LIN {X 0,Y 398.84,Z 465.372,A -85,B 0,C 180,E1 -19980.431,E2 -19980.431} C_VEL
LIN {X 0,Y 402.252,Z 471.24,A -85,B 0,C 180,E1 -19988.433,E2 -19988.433} C_VEL
LIN {X 0,Y 405.408,Z 476.012,A -85,B 0,C 180,E1 -19991.524,E2 -19991.524} C_VEL
LIN {X 0,Y 406.667,Z 477.45,A -85,B 0,C 180,E1 -19992.496,E2 -19992.496} C_VEL
LIN {X 0,Y 410.077,Z 482.026,A -85,B 0,C 180,E1 -19994.834,E2 -19994.834} C_VEL
LIN {X 0,Y 414.526,Z 488.461,A -85,B 0,C 180,E1 -19997.404,E2 -19997.404} C_VEL
LIN {X 0,Y 418.678,Z 494.427,A -85,B 0,C 180,E1 -19999.461,E2 -19999.461} C_VEL
LIN {X 0,Y 424.057,Z 502.276,A -85,B 0,C 180,E1 -20001.8,E2 -20001.8} C_VEL
LIN {X 0,Y 431.293,Z 513.364,A -85,B 0,C 180,E1 -20004.555,E2 -20004.555} C_VEL
LIN {X 0,Y 439.263,Z 526.549,A -85,B 0,C 180,E1 -20007.228,E2 -20007.228} C_VEL
LIN {X 0,Y 440.254,Z 528.583,A -85,B 0,C 180,E1 -20007.551,E2 -20007.551} C_VEL
LIN {X 0,Y 424.232,Z 746.146,A -85,B 0,C 180,E1 -20011.089,E2 -20011.089} C_VEL
LIN {X 0,Y 420.857,Z 772.773,A -85,B 0,C 180,E1 -20011.685,E2 -20011.685} C_VEL
LIN {X 0,Y 417.276,Z 793.387,A -85,B 0,C 180,E1 -20012.304,E2 -20012.304} C_VEL
LIN {X 0,Y 412.24,Z 816.827,A -85,B 0,C 180,E1 -20013.197,E2 -20013.197} C_VEL
LIN {X 0,Y 406.718,Z 837.855,A -85,B 0,C 180,E1 -20014.207,E2 -20014.207} C_VEL
LIN {X 0,Y 400.233,Z 859.541,A -85,B 0,C 180,E1 -20015.469,E2 -20015.469} C_VEL
LIN {X 0,Y 392.916,Z 880.551,A -85,B 0,C 180,E1 -20016.959,E2 -20016.959} C_VEL
LIN {X 0,Y 385.902,Z 898.896,A -85,B 0,C 180,E1 -20018.511,E2 -20018.511} C_VEL
LIN {X 0,Y 376.941,Z 920.104,A -85,B 0,C 180,E1 -20020.654,E2 -20020.654} C_VEL
LIN {X 0,Y 369.253,Z 936.853,A -85,B 0,C 180,E1 -20022.677,E2 -20022.677} C_VEL
LIN {X 0,Y 360.106,Z 955.579,A -85,B 0,C 180,E1 -20025.373,E2 -20025.373} C_VEL
LIN {X 0,Y 352.353,Z 970.558,A -85,B 0,C 180,E1 -20027.956,E2 -20027.956} C_VEL
LIN {X 0,Y 343.98,Z 986.277,A -85,B 0,C 180,E1 -20031.172,E2 -20031.172} C_VEL
LIN {X 0,Y 337.136,Z 998.762,A -85,B 0,C 180,E1 -20034.249,E2 -20034.249} C_VEL
LIN {X 0,Y 330.325,Z 1011.44,A -85,B 0,C 180,E1 -20037.948,E2 -20037.948} C_VEL
LIN {X 0,Y 324.506,Z 1022.333,A -85,B 0,C 180,E1 -20041.873,E2 -20041.873} C_VEL
LIN {X 0,Y 319.832,Z 1031.874,A -85,B 0,C 180,E1 -20046.02,E2 -20046.02} C_VEL
LIN {X 0,Y 316.404,Z 1039.482,A -85,B 0,C 180,E1 -20050.237,E2 -20050.237} C_VEL
LIN {X 0,Y 314.202,Z 1045.368,A -85,B 0,C 180,E1 -20054.306,E2 -20054.306} C_VEL
LIN {X 0,Y 312.792,Z 1050.105,A -85,B 0,C 180,E1 -20058.756,E2 -20058.756} C_VEL
LIN {X 0,Y 312.252,Z 1052.832,A -85,B 0,C 180,E1 -20062.456,E2 -20062.456} C_VEL
LIN {X 0,Y 312.038,Z 1054.512,A -85,B 0,C 180,E1 -20066.142,E2 -20066.142} C_VEL
LIN {X 0,Y 311.99,Z 1055.15,A -85,B 0,C 180,E1 -20070.367,E2 -20070.367} C_VEL
LIN {X 0,Y 312.049,Z 1054.421,A -85,B 0,C 180,E1 -20074.227,E2 -20074.227} C_VEL
LIN {X 0,Y 312.274,Z 1052.681,A -85,B 0,C 180,E1 -20077.914,E2 -20077.914} C_VEL
LIN {X 0,Y 313.002,Z 1049.425,A -85,B 0,C 180,E1 -20082.172,E2 -20082.172} C_VEL
LIN {X 0,Y 314.49,Z 1044.525,A -85,B 0,C 180,E1 -20086.437,E2 -20086.437} C_VEL
LIN {X 0,Y 316.756,Z 1038.711,A -85,B 0,C 180,E1 -20090.359,E2 -20090.359} C_VEL
LIN {X 0,Y 320.659,Z 1030.134,A -85,B 0,C 180,E1 -20094.895,E2 -20094.895} C_VEL
LIN {X 0,Y 324.873,Z 1021.697,A -85,B 0,C 180,E1 -20098.493,E2 -20098.493} C_VEL
LIN {X 0,Y 330.981,Z 1010.268,A -85,B 0,C 180,E1 -20102.53,E2 -20102.53} C_VEL
LIN {X 0,Y 337.538,Z 998.148,A -85,B 0,C 180,E1 -20106.029,E2 -20106.029} C_VEL
LIN {X 0,Y 345.134,Z 984.339,A -85,B 0,C 180,E1 -20109.381,E2 -20109.381} C_VEL
LIN {X 0,Y 353.066,Z 969.367,A -85,B 0,C 180,E1 -20112.378,E2 -20112.378} C_VEL
LIN {X 0,Y 361.534,Z 953.032,A -85,B 0,C 180,E1 -20115.15,E2 -20115.15} C_VEL
LIN {X 0,Y 370.106,Z 935.274,A -85,B 0,C 180,E1 -20117.638,E2 -20117.638} C_VEL
LIN {X 0,Y 378.689,Z 916.559,A -85,B 0,C 180,E1 -20119.853,E2 -20119.853} C_VEL
LIN {X 0,Y 386.864,Z 896.797,A -85,B 0,C 180,E1 -20121.787,E2 -20121.787} C_VEL
LIN {X 0,Y 394.429,Z 876.878,A -85,B 0,C 180,E1 -20123.435,E2 -20123.435} C_VEL
LIN {X 0,Y 401.889,Z 854.633,A -85,B 0,C 180,E1 -20124.94,E2 -20124.94} C_VEL
LIN {X 0,Y 407.945,Z 834.042,A -85,B 0,C 180,E1 -20126.1,E2 -20126.1} C_VEL
LIN {X 0,Y 412.356,Z 817.004,A -85,B 0,C 180,E1 -20126.9,E2 -20126.9} C_VEL
LIN {X 0,Y 413.523,Z 809.94,A -85,B 0,C 180,E1 -20127.317,E2 -20127.317} C_VEL
LIN {X 0,Y 414.052,Z 791.319,A -85,B 0,C 180,E1 -20128.726,E2 -20128.726} C_VEL
LIN {X 0,Y 414.868,Z 785.076,A -85,B 0,C 180,E1 -20129.022,E2 -20129.022} C_VEL
LIN {X 0,Y 418.668,Z 760.478,A -85,B 0,C 180,E1 -20129.662,E2 -20129.662} C_VEL
LIN {X 0,Y 421.165,Z 737.353,A -85,B 0,C 180,E1 -20130.111,E2 -20130.111} C_VEL
LIN {X 0,Y 436.469,Z 532.848,A -85,B 0,C 180,E1 -20133.424,E2 -20133.424} C_VEL
LIN {X 0,Y 428.688,Z 519.811,A -85,B 0,C 180,E1 -20136.129,E2 -20136.129} C_VEL
LIN {X 0,Y 421.455,Z 508.401,A -85,B 0,C 180,E1 -20139.008,E2 -20139.008} C_VEL
LIN {X 0,Y 414.958,Z 498.798,A -85,B 0,C 180,E1 -20142.035,E2 -20142.035} C_VEL
LIN {X 0,Y 411.129,Z 493.354,A -85,B 0,C 180,E1 -20144.121,E2 -20144.121} C_VEL
LIN {X 0,Y 408.284,Z 489.293,A -85,B 0,C 180,E1 -20145.896,E2 -20145.896} C_VEL
LIN {X 0,Y 404.819,Z 484.368,A -85,B 0,C 180,E1 -20148.459,E2 -20148.459} C_VEL
LIN {X 0,Y 401.967,Z 480.55,A -85,B 0,C 180,E1 -20151.128,E2 -20151.128} C_VEL
LIN {X 0,Y 401.27,Z 479.179,A -85,B 0,C 180,E1 -20151.979,E2 -20151.979} C_VEL
LIN {X 0,Y 398.091,Z 474.432,A -85,B 0,C 180,E1 -20159.568,E2 -20159.568} C_VEL
LIN {X 0,Y 398.227,Z 475.335,A -85,B 0,C 180,E1 -20161.871,E2 -20161.871} C_VEL
LIN {X 0,Y 401.485,Z 479.457,A -85,B 0,C 180,E1 -20167.945,E2 -20167.945} C_VEL
LIN {X 0,Y 404.349,Z 483.907,A -85,B 0,C 180,E1 -20170.832,E2 -20170.832} C_VEL
LIN {X 0,Y 405.563,Z 485.403,A -85,B 0,C 180,E1 -20171.808,E2 -20171.808} C_VEL
LIN {X 0,Y 409.4,Z 490.884,A -85,B 0,C 180,E1 -20174.498,E2 -20174.498} C_VEL
LIN {X 0,Y 413.237,Z 496.392,A -85,B 0,C 180,E1 -20176.735,E2 -20176.735} C_VEL
LIN {X 0,Y 417.319,Z 502.3,A -85,B 0,C 180,E1 -20178.8,E2 -20178.8} C_VEL
LIN {X 0,Y 420.643,Z 507.862,A -85,B 0,C 180,E1 -20180.343,E2 -20180.343} C_VEL
LIN {X 0,Y 426.504,Z 518.163,A -85,B 0,C 180,E1 -20182.794,E2 -20182.794} C_VEL
LIN {X 0,Y 434.165,Z 532.67,A -85,B 0,C 180,E1 -20185.62,E2 -20185.62} C_VEL
LIN {X 0,Y 436.3,Z 537.348,A -85,B 0,C 180,E1 -20186.363,E2 -20186.363} C_VEL
LIN {X 0,Y 419.712,Z 757.486,A -85,B 0,C 180,E1 -20189.946,E2 -20189.946} C_VEL
LIN {X 0,Y 416.159,Z 784.326,A -85,B 0,C 180,E1 -20190.522,E2 -20190.522} C_VEL
LIN {X 0,Y 412.096,Z 806.229,A -85,B 0,C 180,E1 -20191.141,E2 -20191.141} C_VEL
LIN {X 0,Y 406.049,Z 832.118,A -85,B 0,C 180,E1 -20192.103,E2 -20192.103} C_VEL
LIN {X 0,Y 400.422,Z 852.323,A -85,B 0,C 180,E1 -20193.057,E2 -20193.057} C_VEL
LIN {X 0,Y 393.151,Z 875.089,A -85,B 0,C 180,E1 -20194.375,E2 -20194.375} C_VEL
LIN {X 0,Y 385.832,Z 895.099,A -85,B 0,C 180,E1 -20195.792,E2 -20195.792} C_VEL
LIN {X 0,Y 377.675,Z 915.487,A -85,B 0,C 180,E1 -20197.512,E2 -20197.512} C_VEL
LIN {X 0,Y 369.176,Z 934.587,A -85,B 0,C 180,E1 -20199.475,E2 -20199.475} C_VEL
LIN {X 0,Y 361.129,Z 951.583,A -85,B 0,C 180,E1 -20201.531,E2 -20201.531} C_VEL
LIN {X 0,Y 351.696,Z 970.23,A -85,B 0,C 180,E1 -20204.238,E2 -20204.238} C_VEL
LIN {X 0,Y 344.137,Z 984.536,A -85,B 0,C 180,E1 -20206.709,E2 -20206.709} C_VEL
LIN {X 0,Y 335.419,Z 1000.614,A -85,B 0,C 180,E1 -20210.007,E2 -20210.007} C_VEL
LIN {X 0,Y 328.07,Z 1013.95,A -85,B 0,C 180,E1 -20213.318,E2 -20213.318} C_VEL
LIN {X 0,Y 321.036,Z 1026.979,A -85,B 0,C 180,E1 -20217.184,E2 -20217.184} C_VEL
LIN {X 0,Y 315.543,Z 1037.501,A -85,B 0,C 180,E1 -20220.999,E2 -20220.999} C_VEL
LIN {X 0,Y 310.872,Z 1047.346,A -85,B 0,C 180,E1 -20225.283,E2 -20225.283} C_VEL
LIN {X 0,Y 307.547,Z 1055.237,A -85,B 0,C 180,E1 -20229.642,E2 -20229.642} C_VEL
LIN {X 0,Y 305.446,Z 1061.626,A -85,B 0,C 180,E1 -20234.039,E2 -20234.039} C_VEL
LIN {X 0,Y 304.32,Z 1066.475,A -85,B 0,C 180,E1 -20238.63,E2 -20238.63} C_VEL
LIN {X 0,Y 303.998,Z 1069.293,A -85,B 0,C 180,E1 -20242.44,E2 -20242.44} C_VEL
LIN {X 0,Y 303.968,Z 1071.08,A -85,B 0,C 180,E1 -20246.417,E2 -20246.417} C_VEL
LIN {X 0,Y 303.99,Z 1071.559,A -85,B 0,C 180,E1 -20250.565,E2 -20250.565} C_VEL
LIN {X 0,Y 303.964,Z 1070.791,A -85,B 0,C 180,E1 -20254.339,E2 -20254.339} C_VEL
LIN {X 0,Y 304.004,Z 1069.044,A -85,B 0,C 180,E1 -20257.94,E2 -20257.94} C_VEL
LIN {X 0,Y 304.413,Z 1065.96,A -85,B 0,C 180,E1 -20261.943,E2 -20261.943} C_VEL
LIN {X 0,Y 305.727,Z 1060.552,A -85,B 0,C 180,E1 -20266.727,E2 -20266.727} C_VEL
LIN {X 0,Y 307.779,Z 1054.575,A -85,B 0,C 180,E1 -20270.739,E2 -20270.739} C_VEL
LIN {X 0,Y 311.571,Z 1045.662,A -85,B 0,C 180,E1 -20275.469,E2 -20275.469} C_VEL
LIN {X 0,Y 316.007,Z 1036.505,A -85,B 0,C 180,E1 -20279.369,E2 -20279.369} C_VEL
LIN {X 0,Y 322.211,Z 1024.682,A -85,B 0,C 180,E1 -20283.53,E2 -20283.53} C_VEL
LIN {X 0,Y 328.76,Z 1012.568,A -85,B 0,C 180,E1 -20287.027,E2 -20287.027} C_VEL
LIN {X 0,Y 336.791,Z 998.007,A -85,B 0,C 180,E1 -20290.555,E2 -20290.555} C_VEL
LIN {X 0,Y 344.827,Z 983.07,A -85,B 0,C 180,E1 -20293.537,E2 -20293.537} C_VEL
LIN {X 0,Y 353.677,Z 966.328,A -85,B 0,C 180,E1 -20296.364,E2 -20296.364} C_VEL
LIN {X 0,Y 362.508,Z 948.447,A -85,B 0,C 180,E1 -20298.851,E2 -20298.851} C_VEL
LIN {X 0,Y 370.86,Z 930.689,A -85,B 0,C 180,E1 -20300.94,E2 -20300.94} C_VEL
LIN {X 0,Y 379.657,Z 910.216,A -85,B 0,C 180,E1 -20302.939,E2 -20302.939} C_VEL
LIN {X 0,Y 387.057,Z 891.531,A -85,B 0,C 180,E1 -20304.463,E2 -20304.463} C_VEL
LIN {X 0,Y 395.358,Z 867.969,A -85,B 0,C 180,E1 -20306.051,E2 -20306.051} C_VEL
LIN {X 0,Y 401.304,Z 848.81,A -85,B 0,C 180,E1 -20307.105,E2 -20307.105} C_VEL
LIN {X 0,Y 407.415,Z 826.398,A -85,B 0,C 180,E1 -20308.121,E2 -20308.121} C_VEL
LIN {X 0,Y 412.484,Z 803.511,A -85,B 0,C 180,E1 -20308.927,E2 -20308.927} C_VEL
LIN {X 0,Y 416.737,Z 779.965,A -85,B 0,C 180,E1 -20309.572,E2 -20309.572} C_VEL
LIN {X 0,Y 419.765,Z 755.051,A -85,B 0,C 180,E1 -20310.084,E2 -20310.084} C_VEL
LIN {X 0,Y 436.13,Z 536.856,A -85,B 0,C 180,E1 -20313.637,E2 -20313.637} C_VEL
LIN {X 0,Y 429.621,Z 524.181,A -85,B 0,C 180,E1 -20315.929,E2 -20315.929} C_VEL
LIN {X 0,Y 423.372,Z 512.779,A -85,B 0,C 180,E1 -20318.381,E2 -20318.381} C_VEL
LIN {X 0,Y 417.521,Z 502.692,A -85,B 0,C 180,E1 -20320.992,E2 -20320.992} C_VEL
LIN {X 0,Y 413.631,Z 497.107,A -85,B 0,C 180,E1 -20322.92,E2 -20322.92} C_VEL
LIN {X 0,Y 411.069,Z 493.426,A -85,B 0,C 180,E1 -20324.336,E2 -20324.336} C_VEL
LIN {X 0,Y 407.99,Z 489,A -85,B 0,C 180,E1 -20326.248,E2 -20326.248} C_VEL
LIN {X 0,Y 404.781,Z 484.386,A -85,B 0,C 180,E1 -20328.602,E2 -20328.602} C_VEL
LIN {X 0,Y 401.616,Z 480.005,A -85,B 0,C 180,E1 -20331.553,E2 -20331.553} C_VEL
LIN {X 0,Y 401.014,Z 479.013,A -85,B 0,C 180,E1 -20332.262,E2 -20332.262} C_VEL
LIN {X 0,Y 397.873,Z 474.137,A -85,B 0,C 180,E1 -20338.848,E2 -20338.848} C_VEL
LIN {X 0,Y 397.864,Z 473.319,A -85,B 0,C 180,E1 -20340.432,E2 -20340.432} C_VEL
LIN {X 0,Y 401.152,Z 479.129,A -85,B 0,C 180,E1 -20348.312,E2 -20348.312} C_VEL
LIN {X 0,Y 404.264,Z 483.898,A -85,B 0,C 180,E1 -20351.412,E2 -20351.412} C_VEL
LIN {X 0,Y 405.406,Z 485.321,A -85,B 0,C 180,E1 -20352.318,E2 -20352.318} C_VEL
LIN {X 0,Y 409.399,Z 490.954,A -85,B 0,C 180,E1 -20355.077,E2 -20355.077} C_VEL
LIN {X 0,Y 413.03,Z 496.212,A -85,B 0,C 180,E1 -20357.178,E2 -20357.178} C_VEL
LIN {X 0,Y 418.41,Z 503.941,A -85,B 0,C 180,E1 -20359.837,E2 -20359.837} C_VEL
LIN {X 0,Y 425.452,Z 514.825,A -85,B 0,C 180,E1 -20362.817,E2 -20362.817} C_VEL
LIN {X 0,Y 432.479,Z 526.228,A -85,B 0,C 180,E1 -20365.396,E2 -20365.396} C_VEL
LIN {X 0,Y 436.287,Z 533.004,A -85,B 0,C 180,E1 -20366.686,E2 -20366.686} C_VEL
LIN {X 0,Y 420.154,Z 746.396,A -85,B 0,C 180,E1 -20370.155,E2 -20370.155} C_VEL
LIN {X 0,Y 416.708,Z 773.001,A -85,B 0,C 180,E1 -20370.748,E2 -20370.748} C_VEL
LIN {X 0,Y 413.075,Z 793.462,A -85,B 0,C 180,E1 -20371.359,E2 -20371.359} C_VEL
LIN {X 0,Y 407.897,Z 817.05,A -85,B 0,C 180,E1 -20372.252,E2 -20372.252} C_VEL
LIN {X 0,Y 402.161,Z 838.378,A -85,B 0,C 180,E1 -20373.275,E2 -20373.275} C_VEL
LIN {X 0,Y 395.294,Z 860.754,A -85,B 0,C 180,E1 -20374.579,E2 -20374.579} C_VEL
LIN {X 0,Y 387.8,Z 881.579,A -85,B 0,C 180,E1 -20376.068,E2 -20376.068} C_VEL
LIN {X 0,Y 380.029,Z 901.307,A -85,B 0,C 180,E1 -20377.755,E2 -20377.755} C_VEL
LIN {X 0,Y 371.133,Z 921.533,A -85,B 0,C 180,E1 -20379.84,E2 -20379.84} C_VEL
LIN {X 0,Y 362.987,Z 938.726,A -85,B 0,C 180,E1 -20381.949,E2 -20381.949} C_VEL
LIN {X 0,Y 353.841,Z 956.717,A -85,B 0,C 180,E1 -20384.594,E2 -20384.594} C_VEL
LIN {X 0,Y 345.862,Z 971.617,A -85,B 0,C 180,E1 -20387.204,E2 -20387.204} C_VEL
LIN {X 0,Y 336.939,Z 987.672,A -85,B 0,C 180,E1 -20390.576,E2 -20390.576} C_VEL
LIN {X 0,Y 330.145,Z 999.611,A -85,B 0,C 180,E1 -20393.586,E2 -20393.586} C_VEL
LIN {X 0,Y 322.986,Z 1012.335,A -85,B 0,C 180,E1 -20397.407,E2 -20397.407} C_VEL
LIN {X 0,Y 317.275,Z 1022.566,A -85,B 0,C 180,E1 -20401.178,E2 -20401.178} C_VEL
LIN {X 0,Y 312.356,Z 1032.094,A -85,B 0,C 180,E1 -20405.409,E2 -20405.409} C_VEL
LIN {X 0,Y 308.722,Z 1039.702,A -85,B 0,C 180,E1 -20409.724,E2 -20409.724} C_VEL
LIN {X 0,Y 306.374,Z 1045.586,A -85,B 0,C 180,E1 -20413.895,E2 -20413.895} C_VEL
LIN {X 0,Y 304.862,Z 1050.321,A -85,B 0,C 180,E1 -20418.459,E2 -20418.459} C_VEL
LIN {X 0,Y 304.276,Z 1053.047,A -85,B 0,C 180,E1 -20422.257,E2 -20422.257} C_VEL
LIN {X 0,Y 304.045,Z 1054.726,A -85,B 0,C 180,E1 -20426.04,E2 -20426.04} C_VEL
LIN {X 0,Y 303.993,Z 1055.363,A -85,B 0,C 180,E1 -20430.377,E2 -20430.377} C_VEL
LIN {X 0,Y 304.056,Z 1054.634,A -85,B 0,C 180,E1 -20434.338,E2 -20434.338} C_VEL
LIN {X 0,Y 304.281,Z 1053.006,A -85,B 0,C 180,E1 -20437.933,E2 -20437.933} C_VEL
LIN {X 0,Y 304.939,Z 1050.106,A -85,B 0,C 180,E1 -20441.922,E2 -20441.922} C_VEL
LIN {X 0,Y 306.595,Z 1044.99,A -85,B 0,C 180,E1 -20446.678,E2 -20446.678} C_VEL
LIN {X 0,Y 308.934,Z 1039.288,A -85,B 0,C 180,E1 -20450.658,E2 -20450.658} C_VEL
LIN {X 0,Y 312.848,Z 1031.149,A -85,B 0,C 180,E1 -20455.156,E2 -20455.156} C_VEL
LIN {X 0,Y 317.426,Z 1022.367,A -85,B 0,C 180,E1 -20459.019,E2 -20459.019} C_VEL
LIN {X 0,Y 323.471,Z 1011.607,A -85,B 0,C 180,E1 -20462.959,E2 -20462.959} C_VEL
LIN {X 0,Y 330.365,Z 999.344,A -85,B 0,C 180,E1 -20466.602,E2 -20466.602} C_VEL
LIN {X 0,Y 338.009,Z 985.993,A -85,B 0,C 180,E1 -20469.936,E2 -20469.936} C_VEL
LIN {X 0,Y 346.544,Z 970.526,A -85,B 0,C 180,E1 -20473.114,E2 -20473.114} C_VEL
LIN {X 0,Y 354.652,Z 955.4,A -85,B 0,C 180,E1 -20475.735,E2 -20475.735} C_VEL
LIN {X 0,Y 363.863,Z 937.14,A -85,B 0,C 180,E1 -20478.37,E2 -20478.37} C_VEL
LIN {X 0,Y 371.824,Z 920.329,A -85,B 0,C 180,E1 -20480.407,E2 -20480.407} C_VEL
LIN {X 0,Y 381.015,Z 899.199,A -85,B 0,C 180,E1 -20482.546,E2 -20482.546} C_VEL
LIN {X 0,Y 388.224,Z 880.852,A -85,B 0,C 180,E1 -20484.097,E2 -20484.097} C_VEL
LIN {X 0,Y 396.047,Z 858.843,A -85,B 0,C 180,E1 -20485.646,E2 -20485.646} C_VEL
LIN {X 0,Y 402.568,Z 837.511,A -85,B 0,C 180,E1 -20486.877,E2 -20486.877} C_VEL
LIN {X 0,Y 408.593,Z 814.944,A -85,B 0,C 180,E1 -20487.945,E2 -20487.945} C_VEL
LIN {X 0,Y 413.602,Z 791.608,A -85,B 0,C 180,E1 -20488.807,E2 -20488.807} C_VEL
LIN {X 0,Y 414.868,Z 785.076,A -85,B 0,C 180,E1 -20489.022,E2 -20489.022} C_VEL
LIN {X 0,Y 415.678,Z 777.754,A -85,B 0,C 180,E1 -20489.363,E2 -20489.363} C_VEL
LIN {X 0,Y 415.335,Z 759.483,A -85,B 0,C 180,E1 -20490.524,E2 -20490.524} C_VEL
LIN {X 0,Y 415.837,Z 752.018,A -85,B 0,C 180,E1 -20490.803,E2 -20490.803} C_VEL
LIN {X 0,Y 419.407,Z 709.213,A -85,B 0,C 180,E1 -20491.53,E2 -20491.53} C_VEL
LIN {X 0,Y 432.567,Z 537.312,A -85,B 0,C 180,E1 -20494.316,E2 -20494.316} C_VEL
LIN {X 0,Y 425.245,Z 524.937,A -85,B 0,C 180,E1 -20496.989,E2 -20496.989} C_VEL
LIN {X 0,Y 418.952,Z 514.929,A -85,B 0,C 180,E1 -20499.607,E2 -20499.607} C_VEL
LIN {X 0,Y 413.188,Z 506.172,A -85,B 0,C 180,E1 -20502.393,E2 -20502.393} C_VEL
LIN {X 0,Y 409.452,Z 500.747,A -85,B 0,C 180,E1 -20504.49,E2 -20504.49} C_VEL
LIN {X 0,Y 406.785,Z 496.87,A -85,B 0,C 180,E1 -20506.206,E2 -20506.206} C_VEL
LIN {X 0,Y 403.499,Z 492.095,A -85,B 0,C 180,E1 -20508.71,E2 -20508.71} C_VEL
LIN {X 0,Y 400.678,Z 488.111,A -85,B 0,C 180,E1 -20511.461,E2 -20511.461} C_VEL
LIN {X 0,Y 400.05,Z 486.996,A -85,B 0,C 180,E1 -20512.243,E2 -20512.243} C_VEL
LIN {X 0,Y 397.115,Z 482.374,A -85,B 0,C 180,E1 -20519.567,E2 -20519.567} C_VEL
LIN {X 0,Y 397.248,Z 483.314,A -85,B 0,C 180,E1 -20521.875,E2 -20521.875} C_VEL
LIN {X 0,Y 400.377,Z 487.415,A -85,B 0,C 180,E1 -20527.823,E2 -20527.823} C_VEL
LIN {X 0,Y 403.208,Z 491.792,A -85,B 0,C 180,E1 -20530.719,E2 -20530.719} C_VEL
LIN {X 0,Y 404.394,Z 493.408,A -85,B 0,C 180,E1 -20531.698,E2 -20531.698} C_VEL
LIN {X 0,Y 407.876,Z 498.429,A -85,B 0,C 180,E1 -20534.191,E2 -20534.191} C_VEL
LIN {X 0,Y 411.628,Z 503.943,A -85,B 0,C 180,E1 -20536.439,E2 -20536.439} C_VEL
LIN {X 0,Y 416.255,Z 510.75,A -85,B 0,C 180,E1 -20538.813,E2 -20538.813} C_VEL
LIN {X 0,Y 423.242,Z 523.257,A -85,B 0,C 180,E1 -20541.954,E2 -20541.954} C_VEL
LIN {X 0,Y 430.627,Z 537.509,A -85,B 0,C 180,E1 -20544.815,E2 -20544.815} C_VEL
LIN {X 0,Y 432.442,Z 541.575,A -85,B 0,C 180,E1 -20545.48,E2 -20545.48} C_VEL
LIN {X 0,Y 415.752,Z 757.4,A -85,B 0,C 180,E1 -20548.989,E2 -20548.989} C_VEL
LIN {X 0,Y 412.138,Z 784.124,A -85,B 0,C 180,E1 -20549.56,E2 -20549.56} C_VEL
LIN {X 0,Y 408.019,Z 805.916,A -85,B 0,C 180,E1 -20550.171,E2 -20550.171} C_VEL
LIN {X 0,Y 402.07,Z 831.01,A -85,B 0,C 180,E1 -20551.091,E2 -20551.091} C_VEL
LIN {X 0,Y 396.315,Z 851.299,A -85,B 0,C 180,E1 -20552.035,E2 -20552.035} C_VEL
LIN {X 0,Y 389.275,Z 873.111,A -85,B 0,C 180,E1 -20553.271,E2 -20553.271} C_VEL
LIN {X 0,Y 381.448,Z 894.071,A -85,B 0,C 180,E1 -20554.737,E2 -20554.737} C_VEL
LIN {X 0,Y 373.304,Z 913.943,A -85,B 0,C 180,E1 -20556.395,E2 -20556.395} C_VEL
LIN {X 0,Y 364.31,Z 933.759,A -85,B 0,C 180,E1 -20558.41,E2 -20558.41} C_VEL
LIN {X 0,Y 356.074,Z 950.663,A -85,B 0,C 180,E1 -20560.448,E2 -20560.448} C_VEL
LIN {X 0,Y 345.996,Z 970.013,A -85,B 0,C 180,E1 -20563.26,E2 -20563.26} C_VEL
LIN {X 0,Y 338.169,Z 984.318,A -85,B 0,C 180,E1 -20565.749,E2 -20565.749} C_VEL
LIN {X 0,Y 329.286,Z 1000.107,A -85,B 0,C 180,E1 -20569.012,E2 -20569.012} C_VEL
LIN {X 0,Y 321.818,Z 1013.087,A -85,B 0,C 180,E1 -20572.26,E2 -20572.26} C_VEL
LIN {X 0,Y 314.654,Z 1025.812,A -85,B 0,C 180,E1 -20576.037,E2 -20576.037} C_VEL
LIN {X 0,Y 308.562,Z 1036.815,A -85,B 0,C 180,E1 -20580.064,E2 -20580.064} C_VEL
LIN {X 0,Y 303.745,Z 1046.326,A -85,B 0,C 180,E1 -20584.245,E2 -20584.245} C_VEL
LIN {X 0,Y 300.09,Z 1054.399,A -85,B 0,C 180,E1 -20588.704,E2 -20588.704} C_VEL
LIN {X 0,Y 297.89,Z 1060.368,A -85,B 0,C 180,E1 -20592.82,E2 -20592.82} C_VEL
LIN {X 0,Y 296.466,Z 1065.765,A -85,B 0,C 180,E1 -20597.732,E2 -20597.732} C_VEL
LIN {X 0,Y 296.016,Z 1068.844,A -85,B 0,C 180,E1 -20601.844,E2 -20601.844} C_VEL
LIN {X 0,Y 295.966,Z 1070.586,A -85,B 0,C 180,E1 -20605.543,E2 -20605.543} C_VEL
LIN {X 0,Y 295.993,Z 1071.349,A -85,B 0,C 180,E1 -20609.419,E2 -20609.419} C_VEL
LIN {X 0,Y 295.969,Z 1070.857,A -85,B 0,C 180,E1 -20613.68,E2 -20613.68} C_VEL
LIN {X 0,Y 295.999,Z 1069.179,A -85,B 0,C 180,E1 -20617.57,E2 -20617.57} C_VEL
LIN {X 0,Y 296.335,Z 1066.401,A -85,B 0,C 180,E1 -20621.483,E2 -20621.483} C_VEL
LIN {X 0,Y 297.444,Z 1061.869,A -85,B 0,C 180,E1 -20626.001,E2 -20626.001} C_VEL
LIN {X 0,Y 299.595,Z 1055.593,A -85,B 0,C 180,E1 -20630.514,E2 -20630.514} C_VEL
LIN {X 0,Y 302.666,Z 1048.514,A -85,B 0,C 180,E1 -20634.598,E2 -20634.598} C_VEL
LIN {X 0,Y 307.826,Z 1038.148,A -85,B 0,C 180,E1 -20639.372,E2 -20639.372} C_VEL
LIN {X 0,Y 313.181,Z 1028.252,A -85,B 0,C 180,E1 -20643.089,E2 -20643.089} C_VEL
LIN {X 0,Y 320.721,Z 1014.918,A -85,B 0,C 180,E1 -20647.216,E2 -20647.216} C_VEL
LIN {X 0,Y 327.616,Z 1002.826,A -85,B 0,C 180,E1 -20650.318,E2 -20650.318} C_VEL
LIN {X 0,Y 336.296,Z 987.588,A -85,B 0,C 180,E1 -20653.613,E2 -20653.613} C_VEL
LIN {X 0,Y 344.957,Z 971.719,A -85,B 0,C 180,E1 -20656.439,E2 -20656.439} C_VEL
LIN {X 0,Y 353.871,Z 954.87,A -85,B 0,C 180,E1 -20658.975,E2 -20658.975} C_VEL
LIN {X 0,Y 363.076,Z 936.086,A -85,B 0,C 180,E1 -20661.307,E2 -20661.307} C_VEL
LIN {X 0,Y 371.37,Z 918.006,A -85,B 0,C 180,E1 -20663.199,E2 -20663.199} C_VEL
LIN {X 0,Y 380.073,Z 897.196,A -85,B 0,C 180,E1 -20665.004,E2 -20665.004} C_VEL
LIN {X 0,Y 387.362,Z 877.906,A -85,B 0,C 180,E1 -20666.395,E2 -20666.395} C_VEL
LIN {X 0,Y 394.927,Z 855.395,A -85,B 0,C 180,E1 -20667.74,E2 -20667.74} C_VEL
LIN {X 0,Y 401.091,Z 833.976,A -85,B 0,C 180,E1 -20668.767,E2 -20668.767} C_VEL
LIN {X 0,Y 406.987,Z 810.111,A -85,B 0,C 180,E1 -20669.685,E2 -20669.685} C_VEL
LIN {X 0,Y 411.572,Z 786.381,A -85,B 0,C 180,E1 -20670.369,E2 -20670.369} C_VEL
LIN {X 0,Y 415.162,Z 761.755,A -85,B 0,C 180,E1 -20670.919,E2 -20670.919} C_VEL
LIN {X 0,Y 419.352,Z 709.809,A -85,B 0,C 180,E1 -20671.793,E2 -20671.793} C_VEL
LIN {X 0,Y 432.274,Z 541.116,A -85,B 0,C 180,E1 -20674.517,E2 -20674.517} C_VEL
LIN {X 0,Y 426.31,Z 529.323,A -85,B 0,C 180,E1 -20676.721,E2 -20676.721} C_VEL
LIN {X 0,Y 420.885,Z 519.274,A -85,B 0,C 180,E1 -20678.941,E2 -20678.941} C_VEL
LIN {X 0,Y 415.687,Z 510.053,A -85,B 0,C 180,E1 -20681.342,E2 -20681.342} C_VEL
LIN {X 0,Y 410.332,Z 501.985,A -85,B 0,C 180,E1 -20684.162,E2 -20684.162} C_VEL
LIN {X 0,Y 406.387,Z 496.447,A -85,B 0,C 180,E1 -20686.627,E2 -20686.627} C_VEL
LIN {X 0,Y 403.453,Z 492.106,A -85,B 0,C 180,E1 -20688.854,E2 -20688.854} C_VEL
LIN {X 0,Y 400.385,Z 487.693,A -85,B 0,C 180,E1 -20691.816,E2 -20691.816} C_VEL
LIN {X 0,Y 399.793,Z 486.814,A -85,B 0,C 180,E1 -20692.527,E2 -20692.527} C_VEL
LIN {X 0,Y 396.879,Z 481.884,A -85,B 0,C 180,E1 -20699.134,E2 -20699.134} C_VEL
LIN {X 0,Y 396.887,Z 481.279,A -85,B 0,C 180,E1 -20700.433,E2 -20700.433} C_VEL
LIN {X 0,Y 399.925,Z 486.94,A -85,B 0,C 180,E1 -20708.049,E2 -20708.049} C_VEL
LIN {X 0,Y 403.295,Z 491.946,A -85,B 0,C 180,E1 -20711.44,E2 -20711.44} C_VEL
LIN {X 0,Y 405.035,Z 494.675,A -85,B 0,C 180,E1 -20712.837,E2 -20712.837} C_VEL
LIN {X 0,Y 407.765,Z 498.323,A -85,B 0,C 180,E1 -20714.702,E2 -20714.702} C_VEL
LIN {X 0,Y 411.42,Z 503.767,A -85,B 0,C 180,E1 -20716.884,E2 -20716.884} C_VEL
LIN {X 0,Y 416.557,Z 511.322,A -85,B 0,C 180,E1 -20719.491,E2 -20719.491} C_VEL
LIN {X 0,Y 423.549,Z 522.348,A -85,B 0,C 180,E1 -20722.522,E2 -20722.522} C_VEL
LIN {X 0,Y 430.735,Z 534.299,A -85,B 0,C 180,E1 -20725.212,E2 -20725.212} C_VEL
LIN {X 0,Y 432.414,Z 537.545,A -85,B 0,C 180,E1 -20725.808,E2 -20725.808} C_VEL
LIN {X 0,Y 416.199,Z 746.549,A -85,B 0,C 180,E1 -20729.201,E2 -20729.201} C_VEL
LIN {X 0,Y 412.692,Z 773.111,A -85,B 0,C 180,E1 -20729.79,E2 -20729.79} C_VEL
LIN {X 0,Y 408.96,Z 793.688,A -85,B 0,C 180,E1 -20730.4,E2 -20730.4} C_VEL
LIN {X 0,Y 403.666,Z 817.273,A -85,B 0,C 180,E1 -20731.288,E2 -20731.288} C_VEL
LIN {X 0,Y 397.956,Z 838.071,A -85,B 0,C 180,E1 -20732.277,E2 -20732.277} C_VEL
LIN {X 0,Y 391.324,Z 859.261,A -85,B 0,C 180,E1 -20733.499,E2 -20733.499} C_VEL
LIN {X 0,Y 383.407,Z 880.993,A -85,B 0,C 180,E1 -20735.027,E2 -20735.027} C_VEL
LIN {X 0,Y 375.719,Z 900.068,A -85,B 0,C 180,E1 -20736.643,E2 -20736.643} C_VEL
LIN {X 0,Y 366.552,Z 920.546,A -85,B 0,C 180,E1 -20738.725,E2 -20738.725} C_VEL
LIN {X 0,Y 358.447,Z 937.206,A -85,B 0,C 180,E1 -20740.749,E2 -20740.749} C_VEL
LIN {X 0,Y 349.16,Z 955.104,A -85,B 0,C 180,E1 -20743.333,E2 -20743.333} C_VEL
LIN {X 0,Y 340.796,Z 970.213,A -85,B 0,C 180,E1 -20745.958,E2 -20745.958} C_VEL
LIN {X 0,Y 332.176,Z 985.372,A -85,B 0,C 180,E1 -20749.073,E2 -20749.073} C_VEL
LIN {X 0,Y 323.939,Z 999.205,A -85,B 0,C 180,E1 -20752.55,E2 -20752.55} C_VEL
LIN {X 0,Y 316.721,Z 1011.513,A -85,B 0,C 180,E1 -20756.246,E2 -20756.246} C_VEL
LIN {X 0,Y 310.366,Z 1022.324,A -85,B 0,C 180,E1 -20760.256,E2 -20760.256} C_VEL
LIN {X 0,Y 305.315,Z 1031.528,A -85,B 0,C 180,E1 -20764.387,E2 -20764.387} C_VEL
LIN {X 0,Y 301.208,Z 1039.624,A -85,B 0,C 180,E1 -20768.991,E2 -20768.991} C_VEL
LIN {X 0,Y 298.743,Z 1045.306,A -85,B 0,C 180,E1 -20773.071,E2 -20773.071} C_VEL
LIN {X 0,Y 296.99,Z 1050.382,A -85,B 0,C 180,E1 -20777.952,E2 -20777.952} C_VEL
LIN {X 0,Y 296.299,Z 1053.262,A -85,B 0,C 180,E1 -20782.047,E2 -20782.047} C_VEL
LIN {X 0,Y 296.051,Z 1054.94,A -85,B 0,C 180,E1 -20785.933,E2 -20785.933} C_VEL
LIN {X 0,Y 295.996,Z 1055.577,A -85,B 0,C 180,E1 -20790.387,E2 -20790.387} C_VEL
LIN {X 0,Y 296.064,Z 1054.848,A -85,B 0,C 180,E1 -20794.455,E2 -20794.455} C_VEL
LIN {X 0,Y 296.303,Z 1053.221,A -85,B 0,C 180,E1 -20798.148,E2 -20798.148} C_VEL
LIN {X 0,Y 297.023,Z 1050.322,A -85,B 0,C 180,E1 -20802.245,E2 -20802.245} C_VEL
LIN {X 0,Y 298.799,Z 1045.207,A -85,B 0,C 180,E1 -20807.126,E2 -20807.126} C_VEL
LIN {X 0,Y 301.294,Z 1039.505,A -85,B 0,C 180,E1 -20811.207,E2 -20811.207} C_VEL
LIN {X 0,Y 305.438,Z 1031.366,A -85,B 0,C 180,E1 -20815.81,E2 -20815.81} C_VEL
LIN {X 0,Y 310.264,Z 1022.585,A -85,B 0,C 180,E1 -20819.755,E2 -20819.755} C_VEL
LIN {X 0,Y 316.831,Z 1011.421,A -85,B 0,C 180,E1 -20823.9,E2 -20823.9} C_VEL
LIN {X 0,Y 323.83,Z 999.515,A -85,B 0,C 180,E1 -20827.482,E2 -20827.482} C_VEL
LIN {X 0,Y 331.756,Z 986.21,A -85,B 0,C 180,E1 -20830.846,E2 -20830.846} C_VEL
LIN {X 0,Y 340.309,Z 971.271,A -85,B 0,C 180,E1 -20833.957,E2 -20833.957} C_VEL
LIN {X 0,Y 348.482,Z 956.533,A -85,B 0,C 180,E1 -20836.546,E2 -20836.546} C_VEL
LIN {X 0,Y 358.225,Z 937.905,A -85,B 0,C 180,E1 -20839.273,E2 -20839.273} C_VEL
LIN {X 0,Y 366.454,Z 921.044,A -85,B 0,C 180,E1 -20841.329,E2 -20841.329} C_VEL
LIN {X 0,Y 375.837,Z 900.141,A -85,B 0,C 180,E1 -20843.461,E2 -20843.461} C_VEL
LIN {X 0,Y 383.222,Z 881.87,A -85,B 0,C 180,E1 -20845.013,E2 -20845.013} C_VEL
LIN {X 0,Y 391.15,Z 860.303,A -85,B 0,C 180,E1 -20846.544,E2 -20846.544} C_VEL
LIN {X 0,Y 398.101,Z 838.142,A -85,B 0,C 180,E1 -20847.825,E2 -20847.825} C_VEL
LIN {X 0,Y 404.361,Z 815.26,A -85,B 0,C 180,E1 -20848.906,E2 -20848.906} C_VEL
LIN {X 0,Y 409.505,Z 791.811,A -85,B 0,C 180,E1 -20849.767,E2 -20849.767} C_VEL
LIN {X 0,Y 413.458,Z 769.612,A -85,B 0,C 180,E1 -20850.407,E2 -20850.407} C_VEL
LIN {X 0,Y 415.837,Z 752.018,A -85,B 0,C 180,E1 -20850.803,E2 -20850.803} C_VEL
LIN {X 0,Y 416.235,Z 744.514,A -85,B 0,C 180,E1 -20851.073,E2 -20851.073} C_VEL
LIN {X 0,Y 414.834,Z 724.825,A -85,B 0,C 180,E1 -20852.159,E2 -20852.159} C_VEL
LIN {X 0,Y 414.962,Z 718.316,A -85,B 0,C 180,E1 -20852.355,E2 -20852.355} C_VEL
LIN {X 0,Y 428.826,Z 541.9,A -85,B 0,C 180,E1 -20855.202,E2 -20855.202} C_VEL
LIN {X 0,Y 421.504,Z 529.451,A -85,B 0,C 180,E1 -20858.024,E2 -20858.024} C_VEL
LIN {X 0,Y 414.771,Z 518.599,A -85,B 0,C 180,E1 -20861.044,E2 -20861.044} C_VEL
LIN {X 0,Y 408.82,Z 509.474,A -85,B 0,C 180,E1 -20864.247,E2 -20864.247} C_VEL
LIN {X 0,Y 405.299,Z 504.444,A -85,B 0,C 180,E1 -20866.518,E2 -20866.518} C_VEL
LIN {X 0,Y 402.187,Z 499.82,A -85,B 0,C 180,E1 -20868.964,E2 -20868.964} C_VEL
LIN {X 0,Y 399.458,Z 495.8,A -85,B 0,C 180,E1 -20871.725,E2 -20871.725} C_VEL
LIN {X 0,Y 398.959,Z 494.883,A -85,B 0,C 180,E1 -20872.367,E2 -20872.367} C_VEL
LIN {X 0,Y 396.14,Z 490.295,A -85,B 0,C 180,E1 -20879.711,E2 -20879.711} C_VEL
LIN {X 0,Y 396.352,Z 491.575,A -85,B 0,C 180,E1 -20882.313,E2 -20882.313} C_VEL
LIN {X 0,Y 399.22,Z 495.236,A -85,B 0,C 180,E1 -20887.628,E2 -20887.628} C_VEL
LIN {X 0,Y 402.069,Z 499.677,A -85,B 0,C 180,E1 -20890.605,E2 -20890.605} C_VEL
LIN {X 0,Y 403.312,Z 501.55,A -85,B 0,C 180,E1 -20891.657,E2 -20891.657} C_VEL
LIN {X 0,Y 406.364,Z 505.973,A -85,B 0,C 180,E1 -20893.881,E2 -20893.881} C_VEL
LIN {X 0,Y 410.03,Z 511.493,A -85,B 0,C 180,E1 -20896.141,E2 -20896.141} C_VEL
LIN {X 0,Y 414.431,Z 518.119,A -85,B 0,C 180,E1 -20898.461,E2 -20898.461} C_VEL
LIN {X 0,Y 421.192,Z 530.585,A -85,B 0,C 180,E1 -20901.59,E2 -20901.59} C_VEL
LIN {X 0,Y 428.323,Z 544.709,A -85,B 0,C 180,E1 -20904.431,E2 -20904.431} C_VEL
LIN {X 0,Y 428.691,Z 545.805,A -85,B 0,C 180,E1 -20904.581,E2 -20904.581} C_VEL
LIN {X 0,Y 411.92,Z 757.206,A -85,B 0,C 180,E1 -20908.012,E2 -20908.012} C_VEL
LIN {X 0,Y 408.235,Z 783.922,A -85,B 0,C 180,E1 -20908.58,E2 -20908.58} C_VEL
LIN {X 0,Y 404.075,Z 805.537,A -85,B 0,C 180,E1 -20909.18,E2 -20909.18} C_VEL
LIN {X 0,Y 398.079,Z 830.403,A -85,B 0,C 180,E1 -20910.08,E2 -20910.08} C_VEL
LIN {X 0,Y 392.432,Z 849.956,A -85,B 0,C 180,E1 -20910.976,E2 -20910.976} C_VEL
LIN {X 0,Y 385.219,Z 871.959,A -85,B 0,C 180,E1 -20912.201,E2 -20912.201} C_VEL
LIN {X 0,Y 377.197,Z 893.043,A -85,B 0,C 180,E1 -20913.657,E2 -20913.657} C_VEL
LIN {X 0,Y 369.181,Z 912.154,A -85,B 0,C 180,E1 -20915.232,E2 -20915.232} C_VEL
LIN {X 0,Y 359.573,Z 932.932,A -85,B 0,C 180,E1 -20917.316,E2 -20917.316} C_VEL
LIN {X 0,Y 351.076,Z 949.887,A -85,B 0,C 180,E1 -20919.353,E2 -20919.353} C_VEL
LIN {X 0,Y 340.926,Z 968.861,A -85,B 0,C 180,E1 -20922.096,E2 -20922.096} C_VEL
LIN {X 0,Y 332.787,Z 983.247,A -85,B 0,C 180,E1 -20924.595,E2 -20924.595} C_VEL
LIN {X 0,Y 323.965,Z 998.464,A -85,B 0,C 180,E1 -20927.713,E2 -20927.713} C_VEL
LIN {X 0,Y 315.572,Z 1012.409,A -85,B 0,C 180,E1 -20931.211,E2 -20931.211} C_VEL
LIN {X 0,Y 308.197,Z 1024.905,A -85,B 0,C 180,E1 -20934.953,E2 -20934.953} C_VEL
LIN {X 0,Y 301.519,Z 1036.39,A -85,B 0,C 180,E1 -20939.193,E2 -20939.193} C_VEL
LIN {X 0,Y 296.52,Z 1045.694,A -85,B 0,C 180,E1 -20943.353,E2 -20943.353} C_VEL
LIN {X 0,Y 292.43,Z 1054.18,A -85,B 0,C 180,E1 -20948.118,E2 -20948.118} C_VEL
LIN {X 0,Y 290.069,Z 1060.15,A -85,B 0,C 180,E1 -20952.341,E2 -20952.341} C_VEL
LIN {X 0,Y 288.524,Z 1065.549,A -85,B 0,C 180,E1 -20957.389,E2 -20957.389} C_VEL
LIN {X 0,Y 288.031,Z 1068.643,A -85,B 0,C 180,E1 -20961.64,E2 -20961.64} C_VEL
LIN {X 0,Y 287.968,Z 1070.372,A -85,B 0,C 180,E1 -20965.419,E2 -20965.419} C_VEL
LIN {X 0,Y 287.996,Z 1071.135,A -85,B 0,C 180,E1 -20969.403,E2 -20969.403} C_VEL
LIN {X 0,Y 287.97,Z 1070.642,A -85,B 0,C 180,E1 -20973.782,E2 -20973.782} C_VEL
LIN {X 0,Y 288.001,Z 1068.964,A -85,B 0,C 180,E1 -20977.782,E2 -20977.782} C_VEL
LIN {X 0,Y 288.382,Z 1066.183,A -85,B 0,C 180,E1 -20981.804,E2 -20981.804} C_VEL
LIN {X 0,Y 289.586,Z 1061.65,A -85,B 0,C 180,E1 -20986.447,E2 -20986.447} C_VEL
LIN {X 0,Y 291.895,Z 1055.373,A -85,B 0,C 180,E1 -20991.08,E2 -20991.08} C_VEL
LIN {X 0,Y 295.166,Z 1048.292,A -85,B 0,C 180,E1 -20995.266,E2 -20995.266} C_VEL
LIN {X 0,Y 300.629,Z 1037.925,A -85,B 0,C 180,E1 -21000.147,E2 -21000.147} C_VEL
LIN {X 0,Y 306.263,Z 1028.029,A -85,B 0,C 180,E1 -21003.937,E2 -21003.937} C_VEL
LIN {X 0,Y 314.319,Z 1014.408,A -85,B 0,C 180,E1 -21008.21,E2 -21008.21} C_VEL
LIN {X 0,Y 321.766,Z 1001.894,A -85,B 0,C 180,E1 -21011.445,E2 -21011.445} C_VEL
LIN {X 0,Y 331.315,Z 985.657,A -85,B 0,C 180,E1 -21014.926,E2 -21014.926} C_VEL
LIN {X 0,Y 339.852,Z 970.562,A -85,B 0,C 180,E1 -21017.602,E2 -21017.602} C_VEL
LIN {X 0,Y 349.649,Z 952.477,A -85,B 0,C 180,E1 -21020.287,E2 -21020.287} C_VEL
LIN {X 0,Y 358.609,Z 934.624,A -85,B 0,C 180,E1 -21022.471,E2 -21022.471} C_VEL
LIN {X 0,Y 367.852,Z 914.939,A -85,B 0,C 180,E1 -21024.498,E2 -21024.498} C_VEL
LIN {X 0,Y 376.515,Z 894.348,A -85,B 0,C 180,E1 -21026.224,E2 -21026.224} C_VEL
LIN {X 0,Y 384.175,Z 874.355,A -85,B 0,C 180,E1 -21027.626,E2 -21027.626} C_VEL
LIN {X 0,Y 391.709,Z 851.768,A -85,B 0,C 180,E1 -21028.915,E2 -21028.915} C_VEL
LIN {X 0,Y 397.688,Z 831.176,A -85,B 0,C 180,E1 -21029.871,E2 -21029.871} C_VEL
LIN {X 0,Y 403.85,Z 805.753,A -85,B 0,C 180,E1 -21030.798,E2 -21030.798} C_VEL
LIN {X 0,Y 408.045,Z 783.969,A -85,B 0,C 180,E1 -21031.404,E2 -21031.404} C_VEL
LIN {X 0,Y 411.738,Z 757.156,A -85,B 0,C 180,E1 -21031.975,E2 -21031.975} C_VEL
LIN {X 0,Y 428.524,Z 545.352,A -85,B 0,C 180,E1 -21035.414,E2 -21035.414} C_VEL
LIN {X 0,Y 421.445,Z 531.308,A -85,B 0,C 180,E1 -21038.204,E2 -21038.204} C_VEL
LIN {X 0,Y 415.274,Z 519.927,A -85,B 0,C 180,E1 -21040.995,E2 -21040.995} C_VEL
LIN {X 0,Y 411.656,Z 513.938,A -85,B 0,C 180,E1 -21042.835,E2 -21042.835} C_VEL
LIN {X 0,Y 407.602,Z 508.055,A -85,B 0,C 180,E1 -21045.146,E2 -21045.146} C_VEL
LIN {X 0,Y 405.003,Z 504.135,A -85,B 0,C 180,E1 -21046.872,E2 -21046.872} C_VEL
LIN {X 0,Y 402.133,Z 499.825,A -85,B 0,C 180,E1 -21049.107,E2 -21049.107} C_VEL
LIN {X 0,Y 399.109,Z 495.248,A -85,B 0,C 180,E1 -21052.152,E2 -21052.152} C_VEL
LIN {X 0,Y 395.913,Z 489.189,A -85,B 0,C 180,E1 -21060.289,E2 -21060.289} C_VEL
LIN {X 0,Y 399.12,Z 495.286,A -85,B 0,C 180,E1 -21068.284,E2 -21068.284} C_VEL
LIN {X 0,Y 401.812,Z 499.5,A -85,B 0,C 180,E1 -21071.047,E2 -21071.047} C_VEL
LIN {X 0,Y 402.899,Z 501.038,A -85,B 0,C 180,E1 -21071.96,E2 -21071.96} C_VEL
LIN {X 0,Y 406.453,Z 506.221,A -85,B 0,C 180,E1 -21074.532,E2 -21074.532} C_VEL
LIN {X 0,Y 409.82,Z 511.321,A -85,B 0,C 180,E1 -21076.586,E2 -21076.586} C_VEL
LIN {X 0,Y 414.788,Z 518.82,A -85,B 0,C 180,E1 -21079.175,E2 -21079.175} C_VEL
LIN {X 0,Y 421.421,Z 529.492,A -85,B 0,C 180,E1 -21082.127,E2 -21082.127} C_VEL
LIN {X 0,Y 428.666,Z 541.8,A -85,B 0,C 180,E1 -21084.909,E2 -21084.909} C_VEL
LIN {X 0,Y 412.351,Z 746.816,A -85,B 0,C 180,E1 -21088.231,E2 -21088.231} C_VEL
LIN {X 0,Y 408.773,Z 773.338,A -85,B 0,C 180,E1 -21088.816,E2 -21088.816} C_VEL
LIN {X 0,Y 404.961,Z 793.913,A -85,B 0,C 180,E1 -21089.421,E2 -21089.421} C_VEL
LIN {X 0,Y 399.553,Z 817.496,A -85,B 0,C 180,E1 -21090.303,E2 -21090.303} C_VEL
LIN {X 0,Y 393.379,Z 839.419,A -85,B 0,C 180,E1 -21091.346,E2 -21091.346} C_VEL
LIN {X 0,Y 386.034,Z 862.112,A -85,B 0,C 180,E1 -21092.669,E2 -21092.669} C_VEL
LIN {X 0,Y 378.181,Z 882.828,A -85,B 0,C 180,E1 -21094.152,E2 -21094.152} C_VEL
LIN {X 0,Y 369.708,Z 903.209,A -85,B 0,C 180,E1 -21095.903,E2 -21095.903} C_VEL
LIN {X 0,Y 360.338,Z 923.183,A -85,B 0,C 180,E1 -21097.996,E2 -21097.996} C_VEL
LIN {X 0,Y 351.187,Z 941.371,A -85,B 0,C 180,E1 -21100.267,E2 -21100.267} C_VEL
LIN {X 0,Y 342.033,Z 958.077,A -85,B 0,C 180,E1 -21102.797,E2 -21102.797} C_VEL
LIN {X 0,Y 333.147,Z 973.592,A -85,B 0,C 180,E1 -21105.588,E2 -21105.588} C_VEL
LIN {X 0,Y 323.995,Z 988.807,A -85,B 0,C 180,E1 -21108.903,E2 -21108.903} C_VEL
LIN {X 0,Y 316.685,Z 1000.681,A -85,B 0,C 180,E1 -21111.998,E2 -21111.998} C_VEL
LIN {X 0,Y 308.606,Z 1013.791,A -85,B 0,C 180,E1 -21116.132,E2 -21116.132} C_VEL
LIN {X 0,Y 302.551,Z 1023.732,A -85,B 0,C 180,E1 -21119.983,E2 -21119.983} C_VEL
LIN {X 0,Y 297.104,Z 1033.231,A -85,B 0,C 180,E1 -21124.483,E2 -21124.483} C_VEL
LIN {X 0,Y 293.29,Z 1040.437,A -85,B 0,C 180,E1 -21128.815,E2 -21128.815} C_VEL
LIN {X 0,Y 290.577,Z 1046.52,A -85,B 0,C 180,E1 -21133.405,E2 -21133.405} C_VEL
LIN {X 0,Y 288.923,Z 1051.065,A -85,B 0,C 180,E1 -21138.218,E2 -21138.218} C_VEL
LIN {X 0,Y 288.289,Z 1053.699,A -85,B 0,C 180,E1 -21142.226,E2 -21142.226} C_VEL
LIN {X 0,Y 288.029,Z 1055.469,A -85,B 0,C 180,E1 -21146.816,E2 -21146.816} C_VEL
LIN {X 0,Y 288.007,Z 1055.701,A -85,B 0,C 180,E1 -21151.194,E2 -21151.194} C_VEL
LIN {X 0,Y 288.087,Z 1054.907,A -85,B 0,C 180,E1 -21155.047,E2 -21155.047} C_VEL
LIN {X 0,Y 288.407,Z 1053.104,A -85,B 0,C 180,E1 -21158.976,E2 -21158.976} C_VEL
LIN {X 0,Y 289.511,Z 1049.33,A -85,B 0,C 180,E1 -21163.951,E2 -21163.951} C_VEL
LIN {X 0,Y 291.337,Z 1044.677,A -85,B 0,C 180,E1 -21168.199,E2 -21168.199} C_VEL
LIN {X 0,Y 294.478,Z 1038.239,A -85,B 0,C 180,E1 -21172.773,E2 -21172.773} C_VEL
LIN {X 0,Y 298.938,Z 1029.991,A -85,B 0,C 180,E1 -21177.274,E2 -21177.274} C_VEL
LIN {X 0,Y 304.339,Z 1020.885,A -85,B 0,C 180,E1 -21181.326,E2 -21181.326} C_VEL
LIN {X 0,Y 311.471,Z 1009.225,A -85,B 0,C 180,E1 -21185.524,E2 -21185.524} C_VEL
LIN {X 0,Y 318.496,Z 997.898,A -85,B 0,C 180,E1 -21188.894,E2 -21188.894} C_VEL
LIN {X 0,Y 327.793,Z 982.702,A -85,B 0,C 180,E1 -21192.624,E2 -21192.624} C_VEL
LIN {X 0,Y 336.293,Z 968.341,A -85,B 0,C 180,E1 -21195.528,E2 -21195.528} C_VEL
LIN {X 0,Y 346.631,Z 950.008,A -85,B 0,C 180,E1 -21198.59,E2 -21198.59} C_VEL
LIN {X 0,Y 354.952,Z 934.264,A -85,B 0,C 180,E1 -21200.775,E2 -21200.775} C_VEL
LIN {X 0,Y 364.678,Z 914.513,A -85,B 0,C 180,E1 -21203.072,E2 -21203.072} C_VEL
LIN {X 0,Y 372.941,Z 895.971,A -85,B 0,C 180,E1 -21204.859,E2 -21204.859} C_VEL
LIN {X 0,Y 381.255,Z 875.598,A -85,B 0,C 180,E1 -21206.511,E2 -21206.511} C_VEL
LIN {X 0,Y 388.835,Z 854.258,A -85,B 0,C 180,E1 -21207.921,E2 -21207.921} C_VEL
LIN {X 0,Y 395.586,Z 832.719,A -85,B 0,C 180,E1 -21209.107,E2 -21209.107} C_VEL
LIN {X 0,Y 401.618,Z 809.643,A -85,B 0,C 180,E1 -21210.121,E2 -21210.121} C_VEL
LIN {X 0,Y 406.405,Z 787.646,A -85,B 0,C 180,E1 -21210.889,E2 -21210.889} C_VEL
LIN {X 0,Y 410.661,Z 762.006,A -85,B 0,C 180,E1 -21211.565,E2 -21211.565} C_VEL
LIN {X 0,Y 413.22,Z 739.786,A -85,B 0,C 180,E1 -21211.999,E2 -21211.999} C_VEL
LIN {X 0,Y 414.962,Z 718.316,A -85,B 0,C 180,E1 -21212.355,E2 -21212.355} C_VEL
LIN {X 0,Y 415.09,Z 710.756,A -85,B 0,C 180,E1 -21212.6,E2 -21212.6} C_VEL
LIN {X 0,Y 413.817,Z 691.073,A -85,B 0,C 180,E1 -21213.693,E2 -21213.693} C_VEL
LIN {X 0,Y 414.007,Z 684.572,A -85,B 0,C 180,E1 -21213.891,E2 -21213.891} C_VEL
LIN {X 0,Y 425.188,Z 546.649,A -85,B 0,C 180,E1 -21216.099,E2 -21216.099} C_VEL
LIN {X 0,Y 418.268,Z 534.662,A -85,B 0,C 180,E1 -21218.913,E2 -21218.913} C_VEL
LIN {X 0,Y 412.351,Z 525.108,A -85,B 0,C 180,E1 -21221.698,E2 -21221.698} C_VEL
LIN {X 0,Y 407.147,Z 516.879,A -85,B 0,C 180,E1 -21224.619,E2 -21224.619} C_VEL
LIN {X 0,Y 403.825,Z 512.016,A -85,B 0,C 180,E1 -21226.833,E2 -21226.833} C_VEL
LIN {X 0,Y 400.883,Z 507.542,A -85,B 0,C 180,E1 -21229.218,E2 -21229.218} C_VEL
LIN {X 0,Y 398.194,Z 503.359,A -85,B 0,C 180,E1 -21232.062,E2 -21232.062} C_VEL
LIN {X 0,Y 397.42,Z 502.438,A -85,B 0,C 180,E1 -21233.064,E2 -21233.064} C_VEL
LIN {X 0,Y 395.164,Z 498.237,A -85,B 0,C 180,E1 -21239.71,E2 -21239.71} C_VEL
LIN {X 0,Y 395.407,Z 499.641,A -85,B 0,C 180,E1 -21242.464,E2 -21242.464} C_VEL
LIN {X 0,Y 398.117,Z 503.185,A -85,B 0,C 180,E1 -21247.504,E2 -21247.504} C_VEL
LIN {X 0,Y 401.097,Z 507.727,A -85,B 0,C 180,E1 -21250.631,E2 -21250.631} C_VEL
LIN {X 0,Y 404.963,Z 513.692,A -85,B 0,C 180,E1 -21253.639,E2 -21253.639} C_VEL
LIN {X 0,Y 408.676,Z 519.412,A -85,B 0,C 180,E1 -21255.977,E2 -21255.977} C_VEL
LIN {X 0,Y 412.819,Z 525.828,A -85,B 0,C 180,E1 -21258.207,E2 -21258.207} C_VEL
LIN {X 0,Y 419.309,Z 538.203,A -85,B 0,C 180,E1 -21261.288,E2 -21261.288} C_VEL
LIN {X 0,Y 425.048,Z 550.012,A -85,B 0,C 180,E1 -21263.666,E2 -21263.666} C_VEL
LIN {X 0,Y 408.209,Z 757.012,A -85,B 0,C 180,E1 -21267.017,E2 -21267.017} C_VEL
LIN {X 0,Y 404.455,Z 783.72,A -85,B 0,C 180,E1 -21267.581,E2 -21267.581} C_VEL
LIN {X 0,Y 400.191,Z 805.449,A -85,B 0,C 180,E1 -21268.179,E2 -21268.179} C_VEL
LIN {X 0,Y 393.958,Z 830.694,A -85,B 0,C 180,E1 -21269.087,E2 -21269.087} C_VEL
LIN {X 0,Y 387.977,Z 850.881,A -85,B 0,C 180,E1 -21270.01,E2 -21270.01} C_VEL
LIN {X 0,Y 380.263,Z 873.596,A -85,B 0,C 180,E1 -21271.287,E2 -21271.287} C_VEL
LIN {X 0,Y 372.413,Z 893.645,A -85,B 0,C 180,E1 -21272.678,E2 -21272.678} C_VEL
LIN {X 0,Y 363.834,Z 913.547,A -85,B 0,C 180,E1 -21274.327,E2 -21274.327} C_VEL
LIN {X 0,Y 354.292,Z 933.46,A -85,B 0,C 180,E1 -21276.347,E2 -21276.347} C_VEL
LIN {X 0,Y 345.34,Z 950.79,A -85,B 0,C 180,E1 -21278.445,E2 -21278.445} C_VEL
LIN {X 0,Y 334.909,Z 969.578,A -85,B 0,C 180,E1 -21281.205,E2 -21281.205} C_VEL
LIN {X 0,Y 326.534,Z 983.882,A -85,B 0,C 180,E1 -21283.725,E2 -21283.725} C_VEL
LIN {X 0,Y 316.973,Z 999.669,A -85,B 0,C 180,E1 -21287.049,E2 -21287.049} C_VEL
LIN {X 0,Y 308.767,Z 1012.805,A -85,B 0,C 180,E1 -21290.419,E2 -21290.419} C_VEL
LIN {X 0,Y 300.761,Z 1025.797,A -85,B 0,C 180,E1 -21294.423,E2 -21294.423} C_VEL
LIN {X 0,Y 294.031,Z 1036.842,A -85,B 0,C 180,E1 -21298.648,E2 -21298.648} C_VEL
LIN {X 0,Y 288.516,Z 1046.686,A -85,B 0,C 180,E1 -21303.222,E2 -21303.222} C_VEL
LIN {X 0,Y 284.507,Z 1054.58,A -85,B 0,C 180,E1 -21307.911,E2 -21307.911} C_VEL
LIN {X 0,Y 281.958,Z 1060.818,A -85,B 0,C 180,E1 -21312.543,E2 -21312.543} C_VEL
LIN {X 0,Y 280.509,Z 1065.661,A -85,B 0,C 180,E1 -21317.441,E2 -21317.441} C_VEL
LIN {X 0,Y 280.034,Z 1068.531,A -85,B 0,C 180,E1 -21321.582,E2 -21321.582} C_VEL
LIN {X 0,Y 279.969,Z 1070.228,A -85,B 0,C 180,E1 -21325.493,E2 -21325.493} C_VEL
LIN {X 0,Y 280.002,Z 1070.968,A -85,B 0,C 180,E1 -21329.795,E2 -21329.795} C_VEL
LIN {X 0,Y 279.969,Z 1070.358,A -85,B 0,C 180,E1 -21334.096,E2 -21334.096} C_VEL
LIN {X 0,Y 280.019,Z 1068.631,A -85,B 0,C 180,E1 -21338.212,E2 -21338.212} C_VEL
LIN {X 0,Y 280.471,Z 1065.795,A -85,B 0,C 180,E1 -21342.359,E2 -21342.359} C_VEL
LIN {X 0,Y 281.906,Z 1060.935,A -85,B 0,C 180,E1 -21347.334,E2 -21347.334} C_VEL
LIN {X 0,Y 284.361,Z 1054.842,A -85,B 0,C 180,E1 -21351.884,E2 -21351.884} C_VEL
LIN {X 0,Y 288.205,Z 1047.164,A -85,B 0,C 180,E1 -21356.478,E2 -21356.478} C_VEL
LIN {X 0,Y 293.753,Z 1037.236,A -85,B 0,C 180,E1 -21361.157,E2 -21361.157} C_VEL
LIN {X 0,Y 299.745,Z 1027.284,A -85,B 0,C 180,E1 -21365.013,E2 -21365.013} C_VEL
LIN {X 0,Y 308.059,Z 1013.828,A -85,B 0,C 180,E1 -21369.266,E2 -21369.266} C_VEL
LIN {X 0,Y 315.603,Z 1001.671,A -85,B 0,C 180,E1 -21372.44,E2 -21372.44} C_VEL
LIN {X 0,Y 325.516,Z 985.434,A -85,B 0,C 180,E1 -21375.954,E2 -21375.954} C_VEL
LIN {X 0,Y 334.348,Z 970.339,A -85,B 0,C 180,E1 -21378.645,E2 -21378.645} C_VEL
LIN {X 0,Y 344.451,Z 952.254,A -85,B 0,C 180,E1 -21381.34,E2 -21381.34} C_VEL
LIN {X 0,Y 353.718,Z 934.311,A -85,B 0,C 180,E1 -21383.535,E2 -21383.535} C_VEL
LIN {X 0,Y 363.081,Z 914.91,A -85,B 0,C 180,E1 -21385.529,E2 -21385.529} C_VEL
LIN {X 0,Y 372.051,Z 894.126,A -85,B 0,C 180,E1 -21387.266,E2 -21387.266} C_VEL
LIN {X 0,Y 379.994,Z 873.86,A -85,B 0,C 180,E1 -21388.678,E2 -21388.678} C_VEL
LIN {X 0,Y 387.596,Z 851.546,A -85,B 0,C 180,E1 -21389.939,E2 -21389.939} C_VEL
LIN {X 0,Y 393.703,Z 830.953,A -85,B 0,C 180,E1 -21390.886,E2 -21390.886} C_VEL
LIN {X 0,Y 399.988,Z 805.531,A -85,B 0,C 180,E1 -21391.804,E2 -21391.804} C_VEL
LIN {X 0,Y 404.239,Z 783.872,A -85,B 0,C 180,E1 -21392.401,E2 -21392.401} C_VEL
LIN {X 0,Y 407.982,Z 757.351,A -85,B 0,C 180,E1 -21392.963,E2 -21392.963} C_VEL
LIN {X 0,Y 420.584,Z 602.178,A -85,B 0,C 180,E1 -21395.489,E2 -21395.489} C_VEL
LIN {X 0,Y 424.829,Z 549.606,A -85,B 0,C 180,E1 -21396.341,E2 -21396.341} C_VEL
LIN {X 0,Y 417.776,Z 535.391,A -85,B 0,C 180,E1 -21399.291,E2 -21399.291} C_VEL
LIN {X 0,Y 411.801,Z 524.381,A -85,B 0,C 180,E1 -21402.185,E2 -21402.185} C_VEL
LIN {X 0,Y 406.844,Z 516.651,A -85,B 0,C 180,E1 -21404.972,E2 -21404.972} C_VEL
LIN {X 0,Y 403.527,Z 511.7,A -85,B 0,C 180,E1 -21407.187,E2 -21407.187} C_VEL
LIN {X 0,Y 400.822,Z 507.541,A -85,B 0,C 180,E1 -21409.362,E2 -21409.362} C_VEL
LIN {X 0,Y 397.61,Z 502.583,A -85,B 0,C 180,E1 -21412.777,E2 -21412.777} C_VEL
LIN {X 0,Y 394.912,Z 497.64,A -85,B 0,C 180,E1 -21419.42,E2 -21419.42} C_VEL
LIN {X 0,Y 394.925,Z 497.256,A -85,B 0,C 180,E1 -21420.435,E2 -21420.435} C_VEL
LIN {X 0,Y 397.96,Z 503.108,A -85,B 0,C 180,E1 -21428.089,E2 -21428.089} C_VEL
LIN {X 0,Y 400.674,Z 507.386,A -85,B 0,C 180,E1 -21430.933,E2 -21430.933} C_VEL
LIN {X 0,Y 402.073,Z 509.63,A -85,B 0,C 180,E1 -21432.131,E2 -21432.131} C_VEL
LIN {X 0,Y 404.944,Z 513.767,A -85,B 0,C 180,E1 -21434.222,E2 -21434.222} C_VEL
LIN {X 0,Y 408.466,Z 519.249,A -85,B 0,C 180,E1 -21436.424,E2 -21436.424} C_VEL
LIN {X 0,Y 413.098,Z 526.432,A -85,B 0,C 180,E1 -21438.889,E2 -21438.889} C_VEL
LIN {X 0,Y 419.937,Z 537.627,A -85,B 0,C 180,E1 -21441.989,E2 -21441.989} C_VEL
LIN {X 0,Y 424.978,Z 546.645,A -85,B 0,C 180,E1 -21444.004,E2 -21444.004} C_VEL
LIN {X 0,Y 408.637,Z 746.945,A -85,B 0,C 180,E1 -21447.24,E2 -21447.24} C_VEL
LIN {X 0,Y 404.974,Z 773.565,A -85,B 0,C 180,E1 -21447.823,E2 -21447.823} C_VEL
LIN {X 0,Y 401.083,Z 794.138,A -85,B 0,C 180,E1 -21448.423,E2 -21448.423} C_VEL
LIN {X 0,Y 395.56,Z 817.718,A -85,B 0,C 180,E1 -21449.298,E2 -21449.298} C_VEL
LIN {X 0,Y 389.253,Z 839.641,A -85,B 0,C 180,E1 -21450.334,E2 -21450.334} C_VEL
LIN {X 0,Y 381.739,Z 862.333,A -85,B 0,C 180,E1 -21451.65,E2 -21451.65} C_VEL
LIN {X 0,Y 373.701,Z 883.049,A -85,B 0,C 180,E1 -21453.126,E2 -21453.126} C_VEL
LIN {X 0,Y 365.012,Z 903.43,A -85,B 0,C 180,E1 -21454.872,E2 -21454.872} C_VEL
LIN {X 0,Y 355.736,Z 922.714,A -85,B 0,C 180,E1 -21456.883,E2 -21456.883} C_VEL
LIN {X 0,Y 346.542,Z 940.492,A -85,B 0,C 180,E1 -21459.09,E2 -21459.09} C_VEL
LIN {X 0,Y 336.53,Z 958.299,A -85,B 0,C 180,E1 -21461.775,E2 -21461.775} C_VEL
LIN {X 0,Y 327.75,Z 973.118,A -85,B 0,C 180,E1 -21464.449,E2 -21464.449} C_VEL
LIN {X 0,Y 317.823,Z 989.08,A -85,B 0,C 180,E1 -21467.943,E2 -21467.943} C_VEL
LIN {X 0,Y 310.252,Z 1000.902,A -85,B 0,C 180,E1 -21471.064,E2 -21471.064} C_VEL
LIN {X 0,Y 301.814,Z 1014.013,A -85,B 0,C 180,E1 -21475.262,E2 -21475.262} C_VEL
LIN {X 0,Y 295.641,Z 1023.668,A -85,B 0,C 180,E1 -21479.064,E2 -21479.064} C_VEL
LIN {X 0,Y 289.942,Z 1033.105,A -85,B 0,C 180,E1 -21483.585,E2 -21483.585} C_VEL
LIN {X 0,Y 285.68,Z 1040.656,A -85,B 0,C 180,E1 -21488.223,E2 -21488.223} C_VEL
LIN {X 0,Y 282.783,Z 1046.738,A -85,B 0,C 180,E1 -21492.934,E2 -21492.934} C_VEL
LIN {X 0,Y 281.008,Z 1051.281,A -85,B 0,C 180,E1 -21497.882,E2 -21497.882} C_VEL
LIN {X 0,Y 280.315,Z 1053.914,A -85,B 0,C 180,E1 -21502.004,E2 -21502.004} C_VEL
LIN {X 0,Y 280.035,Z 1055.683,A -85,B 0,C 180,E1 -21506.725,E2 -21506.725} C_VEL
LIN {X 0,Y 280.01,Z 1055.914,A -85,B 0,C 180,E1 -21511.228,E2 -21511.228} C_VEL
LIN {X 0,Y 280.094,Z 1055.14,A -85,B 0,C 180,E1 -21515.132,E2 -21515.132} C_VEL
LIN {X 0,Y 280.451,Z 1053.319,A -85,B 0,C 180,E1 -21519.232,E2 -21519.232} C_VEL
LIN {X 0,Y 281.655,Z 1049.508,A -85,B 0,C 180,E1 -21524.389,E2 -21524.389} C_VEL
LIN {X 0,Y 283.6,Z 1044.894,A -85,B 0,C 180,E1 -21528.714,E2 -21528.714} C_VEL
LIN {X 0,Y 286.943,Z 1038.457,A -85,B 0,C 180,E1 -21533.406,E2 -21533.406} C_VEL
LIN {X 0,Y 291.661,Z 1030.209,A -85,B 0,C 180,E1 -21538.013,E2 -21538.013} C_VEL
LIN {X 0,Y 297.271,Z 1021.214,A -85,B 0,C 180,E1 -21542.103,E2 -21542.103} C_VEL
LIN {X 0,Y 304.816,Z 1009.442,A -85,B 0,C 180,E1 -21546.423,E2 -21546.423} C_VEL
LIN {X 0,Y 312.144,Z 998.115,A -85,B 0,C 180,E1 -21549.841,E2 -21549.841} C_VEL
LIN {X 0,Y 321.822,Z 982.887,A -85,B 0,C 180,E1 -21553.62,E2 -21553.62} C_VEL
LIN {X 0,Y 330.609,Z 968.557,A -85,B 0,C 180,E1 -21556.54,E2 -21556.54} C_VEL
LIN {X 0,Y 341.288,Z 950.222,A -85,B 0,C 180,E1 -21559.618,E2 -21559.618} C_VEL
LIN {X 0,Y 349.86,Z 934.477,A -85,B 0,C 180,E1 -21561.808,E2 -21561.808} C_VEL
LIN {X 0,Y 359.862,Z 914.712,A -85,B 0,C 180,E1 -21564.107,E2 -21564.107} C_VEL
LIN {X 0,Y 368.338,Z 896.182,A -85,B 0,C 180,E1 -21565.889,E2 -21565.889} C_VEL
LIN {X 0,Y 376.86,Z 875.808,A -85,B 0,C 180,E1 -21567.535,E2 -21567.535} C_VEL
LIN {X 0,Y 384.614,Z 854.467,A -85,B 0,C 180,E1 -21568.938,E2 -21568.938} C_VEL
LIN {X 0,Y 391.519,Z 832.927,A -85,B 0,C 180,E1 -21570.117,E2 -21570.117} C_VEL
LIN {X 0,Y 397.681,Z 809.841,A -85,B 0,C 180,E1 -21571.124,E2 -21571.124} C_VEL
LIN {X 0,Y 402.517,Z 788.083,A -85,B 0,C 180,E1 -21571.878,E2 -21571.878} C_VEL
LIN {X 0,Y 406.886,Z 762.364,A -85,B 0,C 180,E1 -21572.553,E2 -21572.553} C_VEL
LIN {X 0,Y 409.51,Z 740.107,A -85,B 0,C 180,E1 -21572.986,E2 -21572.986} C_VEL
LIN {X 0,Y 414.007,Z 684.572,A -85,B 0,C 180,E1 -21573.891,E2 -21573.891} C_VEL
LIN {X 0,Y 414.181,Z 677.014,A -85,B 0,C 180,E1 -21574.136,E2 -21574.136} C_VEL
LIN {X 0,Y 413.111,Z 657.341,A -85,B 0,C 180,E1 -21575.239,E2 -21575.239} C_VEL
LIN {X 0,Y 413.33,Z 650.843,A -85,B 0,C 180,E1 -21575.44,E2 -21575.44} C_VEL
LIN {X 0,Y 421.602,Z 551.341,A -85,B 0,C 180,E1 -21577.03,E2 -21577.03} C_VEL
LIN {X 0,Y 415.552,Z 540.719,A -85,B 0,C 180,E1 -21579.617,E2 -21579.617} C_VEL
LIN {X 0,Y 409.8,Z 531.284,A -85,B 0,C 180,E1 -21582.462,E2 -21582.462} C_VEL
LIN {X 0,Y 405.163,Z 523.837,A -85,B 0,C 180,E1 -21585.201,E2 -21585.201} C_VEL
LIN {X 0,Y 402.364,Z 519.587,A -85,B 0,C 180,E1 -21587.149,E2 -21587.149} C_VEL
LIN {X 0,Y 399.588,Z 515.262,A -85,B 0,C 180,E1 -21589.475,E2 -21589.475} C_VEL
LIN {X 0,Y 396.992,Z 511.048,A -85,B 0,C 180,E1 -21592.329,E2 -21592.329} C_VEL
LIN {X 0,Y 394.189,Z 506.179,A -85,B 0,C 180,E1 -21599.709,E2 -21599.709} C_VEL
LIN {X 0,Y 394.463,Z 507.727,A -85,B 0,C 180,E1 -21602.615,E2 -21602.615} C_VEL
LIN {X 0,Y 396.968,Z 511,A -85,B 0,C 180,E1 -21607.308,E2 -21607.308} C_VEL
LIN {X 0,Y 400.42,Z 516.492,A -85,B 0,C 180,E1 -21610.94,E2 -21610.94} C_VEL
LIN {X 0,Y 403.568,Z 521.409,A -85,B 0,C 180,E1 -21613.395,E2 -21613.395} C_VEL
LIN {X 0,Y 407.211,Z 527.141,A -85,B 0,C 180,E1 -21615.743,E2 -21615.743} C_VEL
LIN {X 0,Y 411.079,Z 533.371,A -85,B 0,C 180,E1 -21617.884,E2 -21617.884} C_VEL
LIN {X 0,Y 417.146,Z 545.226,A -85,B 0,C 180,E1 -21620.852,E2 -21620.852} C_VEL
LIN {X 0,Y 421.488,Z 554.536,A -85,B 0,C 180,E1 -21622.741,E2 -21622.741} C_VEL
LIN {X 0,Y 404.625,Z 756.819,A -85,B 0,C 180,E1 -21626.003,E2 -21626.003} C_VEL
LIN {X 0,Y 400.8,Z 783.518,A -85,B 0,C 180,E1 -21626.563,E2 -21626.563} C_VEL
LIN {X 0,Y 396.482,Z 805.13,A -85,B 0,C 180,E1 -21627.151,E2 -21627.151} C_VEL
LIN {X 0,Y 390.245,Z 830.001,A -85,B 0,C 180,E1 -21628.032,E2 -21628.032} C_VEL
LIN {X 0,Y 384.358,Z 849.537,A -85,B 0,C 180,E1 -21628.909,E2 -21628.909} C_VEL
LIN {X 0,Y 376.82,Z 871.538,A -85,B 0,C 180,E1 -21630.113,E2 -21630.113} C_VEL
LIN {X 0,Y 368.425,Z 892.618,A -85,B 0,C 180,E1 -21631.55,E2 -21631.55} C_VEL
LIN {X 0,Y 359.951,Z 911.856,A -85,B 0,C 180,E1 -21633.12,E2 -21633.12} C_VEL
LIN {X 0,Y 349.88,Z 932.501,A -85,B 0,C 180,E1 -21635.181,E2 -21635.181} C_VEL
LIN {X 0,Y 340.891,Z 949.456,A -85,B 0,C 180,E1 -21637.216,E2 -21637.216} C_VEL
LIN {X 0,Y 330.096,Z 968.427,A -85,B 0,C 180,E1 -21639.972,E2 -21639.972} C_VEL
LIN {X 0,Y 321.395,Z 982.811,A -85,B 0,C 180,E1 -21642.495,E2 -21642.495} C_VEL
LIN {X 0,Y 311.916,Z 998.027,A -85,B 0,C 180,E1 -21645.667,E2 -21645.667} C_VEL
LIN {X 0,Y 302.945,Z 1011.786,A -85,B 0,C 180,E1 -21649.193,E2 -21649.193} C_VEL
LIN {X 0,Y 295.119,Z 1023.884,A -85,B 0,C 180,E1 -21652.909,E2 -21652.909} C_VEL
LIN {X 0,Y 287.566,Z 1035.689,A -85,B 0,C 180,E1 -21657.388,E2 -21657.388} C_VEL
LIN {X 0,Y 282.055,Z 1044.842,A -85,B 0,C 180,E1 -21661.638,E2 -21661.638} C_VEL
LIN {X 0,Y 277.202,Z 1053.742,A -85,B 0,C 180,E1 -21666.848,E2 -21666.848} C_VEL
LIN {X 0,Y 274.481,Z 1059.713,A -85,B 0,C 180,E1 -21671.302,E2 -21671.302} C_VEL
LIN {X 0,Y 272.662,Z 1065.115,A -85,B 0,C 180,E1 -21676.642,E2 -21676.642} C_VEL
LIN {X 0,Y 272.062,Z 1068.199,A -85,B 0,C 180,E1 -21681.12,E2 -21681.12} C_VEL
LIN {X 0,Y 271.972,Z 1069.944,A -85,B 0,C 180,E1 -21685.149,E2 -21685.149} C_VEL
LIN {X 0,Y 272.001,Z 1070.685,A -85,B 0,C 180,E1 -21689.157,E2 -21689.157} C_VEL
LIN {X 0,Y 271.975,Z 1070.353,A -85,B 0,C 180,E1 -21693.583,E2 -21693.583} C_VEL
LIN {X 0,Y 272.021,Z 1068.532,A -85,B 0,C 180,E1 -21698.242,E2 -21698.242} C_VEL
LIN {X 0,Y 272.492,Z 1065.749,A -85,B 0,C 180,E1 -21702.503,E2 -21702.503} C_VEL
LIN {X 0,Y 273.915,Z 1061.211,A -85,B 0,C 180,E1 -21707.417,E2 -21707.417} C_VEL
LIN {X 0,Y 276.583,Z 1054.931,A -85,B 0,C 180,E1 -21712.308,E2 -21712.308} C_VEL
LIN {X 0,Y 280.293,Z 1047.848,A -85,B 0,C 180,E1 -21716.71,E2 -21716.71} C_VEL
LIN {X 0,Y 286.406,Z 1037.48,A -85,B 0,C 180,E1 -21721.814,E2 -21721.814} C_VEL
LIN {X 0,Y 292.643,Z 1027.583,A -85,B 0,C 180,E1 -21725.751,E2 -21725.751} C_VEL
LIN {X 0,Y 301.273,Z 1014.248,A -85,B 0,C 180,E1 -21730.08,E2 -21730.08} C_VEL
LIN {X 0,Y 309.08,Z 1002.156,A -85,B 0,C 180,E1 -21733.301,E2 -21733.301} C_VEL
LIN {X 0,Y 318.802,Z 986.918,A -85,B 0,C 180,E1 -21736.689,E2 -21736.689} C_VEL
LIN {X 0,Y 328.413,Z 971.032,A -85,B 0,C 180,E1 -21739.571,E2 -21739.571} C_VEL
LIN {X 0,Y 338.503,Z 953.661,A -85,B 0,C 180,E1 -21742.207,E2 -21742.207} C_VEL
LIN {X 0,Y 348.594,Z 934.701,A -85,B 0,C 180,E1 -21744.549,E2 -21744.549} C_VEL
LIN {X 0,Y 357.949,Z 915.856,A -85,B 0,C 180,E1 -21746.494,E2 -21746.494} C_VEL
LIN {X 0,Y 367.371,Z 894.719,A -85,B 0,C 180,E1 -21748.271,E2 -21748.271} C_VEL
LIN {X 0,Y 375.025,Z 875.719,A -85,B 0,C 180,E1 -21749.6,E2 -21749.6} C_VEL
LIN {X 0,Y 383.247,Z 852.458,A -85,B 0,C 180,E1 -21750.928,E2 -21750.928} C_VEL
LIN {X 0,Y 389.469,Z 832.019,A -85,B 0,C 180,E1 -21751.869,E2 -21751.869} C_VEL
LIN {X 0,Y 395.777,Z 807.479,A -85,B 0,C 180,E1 -21752.764,E2 -21752.764} C_VEL
LIN {X 0,Y 400.318,Z 785.082,A -85,B 0,C 180,E1 -21753.384,E2 -21753.384} C_VEL
LIN {X 0,Y 404.092,Z 760.121,A -85,B 0,C 180,E1 -21753.924,E2 -21753.924} C_VEL
LIN {X 0,Y 409.049,Z 702.462,A -85,B 0,C 180,E1 -21754.881,E2 -21754.881} C_VEL
LIN {X 0,Y 421.257,Z 553.983,A -85,B 0,C 180,E1 -21757.275,E2 -21757.275} C_VEL
LIN {X 0,Y 415.143,Z 541.47,A -85,B 0,C 180,E1 -21759.964,E2 -21759.964} C_VEL
LIN {X 0,Y 410.021,Z 531.741,A -85,B 0,C 180,E1 -21762.545,E2 -21762.545} C_VEL
LIN {X 0,Y 405.298,Z 524.197,A -85,B 0,C 180,E1 -21765.279,E2 -21765.279} C_VEL
LIN {X 0,Y 401.97,Z 519.138,A -85,B 0,C 180,E1 -21767.575,E2 -21767.575} C_VEL
LIN {X 0,Y 399.518,Z 515.256,A -85,B 0,C 180,E1 -21769.619,E2 -21769.619} C_VEL
LIN {X 0,Y 396.521,Z 510.468,A -85,B 0,C 180,E1 -21772.902,E2 -21772.902} C_VEL
LIN {X 0,Y 393.933,Z 505.517,A -85,B 0,C 180,E1 -21779.564,E2 -21779.564} C_VEL
LIN {X 0,Y 393.944,Z 505.249,A -85,B 0,C 180,E1 -21780.436,E2 -21780.436} C_VEL
LIN {X 0,Y 396.856,Z 511.062,A -85,B 0,C 180,E1 -21787.965,E2 -21787.965} C_VEL
LIN {X 0,Y 399.538,Z 515.271,A -85,B 0,C 180,E1 -21790.818,E2 -21790.818} C_VEL
LIN {X 0,Y 403.545,Z 521.484,A -85,B 0,C 180,E1 -21793.98,E2 -21793.98} C_VEL
LIN {X 0,Y 407,Z 526.984,A -85,B 0,C 180,E1 -21796.191,E2 -21796.191} C_VEL
LIN {X 0,Y 411.616,Z 534.382,A -85,B 0,C 180,E1 -21798.702,E2 -21798.702} C_VEL
LIN {X 0,Y 417.985,Z 545.058,A -85,B 0,C 180,E1 -21801.654,E2 -21801.654} C_VEL
LIN {X 0,Y 421.408,Z 551.366,A -85,B 0,C 180,E1 -21803.081,E2 -21803.081} C_VEL
LIN {X 0,Y 405.037,Z 747.181,A -85,B 0,C 180,E1 -21806.234,E2 -21806.234} C_VEL
LIN {X 0,Y 401.32,Z 773.676,A -85,B 0,C 180,E1 -21806.809,E2 -21806.809} C_VEL
LIN {X 0,Y 397.341,Z 794.308,A -85,B 0,C 180,E1 -21807.405,E2 -21807.405} C_VEL
LIN {X 0,Y 391.691,Z 817.941,A -85,B 0,C 180,E1 -21808.273,E2 -21808.273} C_VEL
LIN {X 0,Y 385.251,Z 839.863,A -85,B 0,C 180,E1 -21809.301,E2 -21809.301} C_VEL
LIN {X 0,Y 377.569,Z 862.555,A -85,B 0,C 180,E1 -21810.608,E2 -21810.608} C_VEL
LIN {X 0,Y 369.346,Z 883.27,A -85,B 0,C 180,E1 -21812.076,E2 -21812.076} C_VEL
LIN {X 0,Y 360.483,Z 903.553,A -85,B 0,C 180,E1 -21813.806,E2 -21813.806} C_VEL
LIN {X 0,Y 350.875,Z 923.021,A -85,B 0,C 180,E1 -21815.832,E2 -21815.832} C_VEL
LIN {X 0,Y 341.463,Z 940.713,A -85,B 0,C 180,E1 -21818.029,E2 -21818.029} C_VEL
LIN {X 0,Y 331.138,Z 958.52,A -85,B 0,C 180,E1 -21820.72,E2 -21820.72} C_VEL
LIN {X 0,Y 321.557,Z 974.176,A -85,B 0,C 180,E1 -21823.571,E2 -21823.571} C_VEL
LIN {X 0,Y 311.812,Z 989.25,A -85,B 0,C 180,E1 -21826.919,E2 -21826.919} C_VEL
LIN {X 0,Y 303.906,Z 1001.123,A -85,B 0,C 180,E1 -21830.091,E2 -21830.091} C_VEL
LIN {X 0,Y 295.094,Z 1014.234,A -85,B 0,C 180,E1 -21834.352,E2 -21834.352} C_VEL
LIN {X 0,Y 288.625,Z 1023.889,A -85,B 0,C 180,E1 -21838.226,E2 -21838.226} C_VEL
LIN {X 0,Y 282.617,Z 1033.325,A -85,B 0,C 180,E1 -21842.845,E2 -21842.845} C_VEL
LIN {X 0,Y 278.1,Z 1040.876,A -85,B 0,C 180,E1 -21847.597,E2 -21847.597} C_VEL
LIN {X 0,Y 274.904,Z 1047.189,A -85,B 0,C 180,E1 -21852.647,E2 -21852.647} C_VEL
LIN {X 0,Y 273.099,Z 1051.498,A -85,B 0,C 180,E1 -21857.525,E2 -21857.525} C_VEL
LIN {X 0,Y 272.322,Z 1054.24,A -85,B 0,C 180,E1 -21861.98,E2 -21861.98} C_VEL
LIN {X 0,Y 272.034,Z 1055.919,A -85,B 0,C 180,E1 -21866.84,E2 -21866.84} C_VEL
LIN {X 0,Y 272.013,Z 1056.127,A -85,B 0,C 180,E1 -21871.264,E2 -21871.264} C_VEL
LIN {X 0,Y 272.103,Z 1055.358,A -85,B 0,C 180,E1 -21875.271,E2 -21875.271} C_VEL
LIN {X 0,Y 272.498,Z 1053.534,A -85,B 0,C 180,E1 -21879.504,E2 -21879.504} C_VEL
LIN {X 0,Y 273.797,Z 1049.724,A -85,B 0,C 180,E1 -21884.811,E2 -21884.811} C_VEL
LIN {X 0,Y 275.886,Z 1045.111,A -85,B 0,C 180,E1 -21889.257,E2 -21889.257} C_VEL
LIN {X 0,Y 279.574,Z 1038.469,A -85,B 0,C 180,E1 -21894.216,E2 -21894.216} C_VEL
LIN {X 0,Y 284.726,Z 1029.971,A -85,B 0,C 180,E1 -21899.022,E2 -21899.022} C_VEL
LIN {X 0,Y 291.287,Z 1020.076,A -85,B 0,C 180,E1 -21903.55,E2 -21903.55} C_VEL
LIN {X 0,Y 298.994,Z 1008.529,A -85,B 0,C 180,E1 -21907.733,E2 -21907.733} C_VEL
LIN {X 0,Y 307.619,Z 995.824,A -85,B 0,C 180,E1 -21911.536,E2 -21911.536} C_VEL
LIN {X 0,Y 316.889,Z 981.61,A -85,B 0,C 180,E1 -21914.975,E2 -21914.975} C_VEL
LIN {X 0,Y 326.105,Z 967.098,A -85,B 0,C 180,E1 -21917.903,E2 -21917.903} C_VEL
LIN {X 0,Y 336.343,Z 949.934,A -85,B 0,C 180,E1 -21920.753,E2 -21920.753} C_VEL
LIN {X 0,Y 344.885,Z 934.691,A -85,B 0,C 180,E1 -21922.871,E2 -21922.871} C_VEL
LIN {X 0,Y 354.926,Z 915.418,A -85,B 0,C 180,E1 -21925.118,E2 -21925.118} C_VEL
LIN {X 0,Y 363.661,Z 896.826,A -85,B 0,C 180,E1 -21926.907,E2 -21926.907} C_VEL
LIN {X 0,Y 372.588,Z 876.018,A -85,B 0,C 180,E1 -21928.583,E2 -21928.583} C_VEL
LIN {X 0,Y 380.519,Z 854.676,A -85,B 0,C 180,E1 -21929.978,E2 -21929.978} C_VEL
LIN {X 0,Y 387.447,Z 833.533,A -85,B 0,C 180,E1 -21931.128,E2 -21931.128} C_VEL
LIN {X 0,Y 393.669,Z 810.856,A -85,B 0,C 180,E1 -21932.116,E2 -21932.116} C_VEL
LIN {X 0,Y 398.572,Z 789.369,A -85,B 0,C 180,E1 -21932.86,E2 -21932.86} C_VEL
LIN {X 0,Y 403.213,Z 762.885,A -85,B 0,C 180,E1 -21933.556,E2 -21933.556} C_VEL
LIN {X 0,Y 405.896,Z 740.703,A -85,B 0,C 180,E1 -21933.985,E2 -21933.985} C_VEL
LIN {X 0,Y 413.33,Z 650.843,A -85,B 0,C 180,E1 -21935.44,E2 -21935.44} C_VEL
LIN {X 0,Y 413.54,Z 643.287,A -85,B 0,C 180,E1 -21935.688,E2 -21935.688} C_VEL
LIN {X 0,Y 412.679,Z 623.619,A -85,B 0,C 180,E1 -21936.798,E2 -21936.798} C_VEL
LIN {X 0,Y 412.944,Z 617.12,A -85,B 0,C 180,E1 -21936.995,E2 -21936.995} C_VEL
LIN {X 0,Y 418.104,Z 556.051,A -85,B 0,C 180,E1 -21937.984,E2 -21937.984} C_VEL
LIN {X 0,Y 412.687,Z 546.458,A -85,B 0,C 180,E1 -21940.43,E2 -21940.43} C_VEL
LIN {X 0,Y 407.593,Z 537.866,A -85,B 0,C 180,E1 -21943.084,E2 -21943.084} C_VEL
LIN {X 0,Y 403.328,Z 530.926,A -85,B 0,C 180,E1 -21945.719,E2 -21945.719} C_VEL
LIN {X 0,Y 400.915,Z 527.155,A -85,B 0,C 180,E1 -21947.468,E2 -21947.468} C_VEL
LIN {X 0,Y 398.3,Z 522.98,A -85,B 0,C 180,E1 -21949.733,E2 -21949.733} C_VEL
LIN {X 0,Y 395.586,Z 518.463,A -85,B 0,C 180,E1 -21952.885,E2 -21952.885} C_VEL
LIN {X 0,Y 393.216,Z 514.1,A -85,B 0,C 180,E1 -21959.854,E2 -21959.854} C_VEL
LIN {X 0,Y 395.873,Z 518.938,A -85,B 0,C 180,E1 -21967.182,E2 -21967.182} C_VEL
LIN {X 0,Y 399.111,Z 524.185,A -85,B 0,C 180,E1 -21970.684,E2 -21970.684} C_VEL
LIN {X 0,Y 402.182,Z 529.123,A -85,B 0,C 180,E1 -21973.149,E2 -21973.149} C_VEL
LIN {X 0,Y 405.64,Z 534.687,A -85,B 0,C 180,E1 -21975.439,E2 -21975.439} C_VEL
LIN {X 0,Y 409.231,Z 540.646,A -85,B 0,C 180,E1 -21977.49,E2 -21977.49} C_VEL
LIN {X 0,Y 414.984,Z 552.197,A -85,B 0,C 180,E1 -21980.4,E2 -21980.4} C_VEL
LIN {X 0,Y 418.04,Z 559.067,A -85,B 0,C 180,E1 -21981.8,E2 -21981.8} C_VEL
LIN {X 0,Y 401.169,Z 756.625,A -85,B 0,C 180,E1 -21984.972,E2 -21984.972} C_VEL
LIN {X 0,Y 397.273,Z 783.317,A -85,B 0,C 180,E1 -21985.527,E2 -21985.527} C_VEL
LIN {X 0,Y 392.889,Z 804.876,A -85,B 0,C 180,E1 -21986.106,E2 -21986.106} C_VEL
LIN {X 0,Y 386.522,Z 829.793,A -85,B 0,C 180,E1 -21986.978,E2 -21986.978} C_VEL
LIN {X 0,Y 380.515,Z 849.328,A -85,B 0,C 180,E1 -21987.843,E2 -21987.843} C_VEL
LIN {X 0,Y 372.721,Z 871.586,A -85,B 0,C 180,E1 -21989.05,E2 -21989.05} C_VEL
LIN {X 0,Y 363.883,Z 893.222,A -85,B 0,C 180,E1 -21990.521,E2 -21990.521} C_VEL
LIN {X 0,Y 354.545,Z 913.859,A -85,B 0,C 180,E1 -21992.214,E2 -21992.214} C_VEL
LIN {X 0,Y 344.576,Z 933.511,A -85,B 0,C 180,E1 -21994.207,E2 -21994.207} C_VEL
LIN {X 0,Y 335.061,Z 950.917,A -85,B 0,C 180,E1 -21996.318,E2 -21996.318} C_VEL
LIN {X 0,Y 324.283,Z 969.144,A -85,B 0,C 180,E1 -21999.012,E2 -21999.012} C_VEL
LIN {X 0,Y 315.333,Z 983.446,A -85,B 0,C 180,E1 -22001.554,E2 -22001.554} C_VEL
LIN {X 0,Y 305.064,Z 999.232,A -85,B 0,C 180,E1 -22004.93,E2 -22004.93} C_VEL
LIN {X 0,Y 296.282,Z 1012.21,A -85,B 0,C 180,E1 -22008.33,E2 -22008.33} C_VEL
LIN {X 0,Y 287.794,Z 1024.823,A -85,B 0,C 180,E1 -22012.303,E2 -22012.303} C_VEL
LIN {X 0,Y 280.307,Z 1035.935,A -85,B 0,C 180,E1 -22016.678,E2 -22016.678} C_VEL
LIN {X 0,Y 274.316,Z 1045.447,A -85,B 0,C 180,E1 -22021.24,E2 -22021.24} C_VEL
LIN {X 0,Y 269.47,Z 1053.832,A -85,B 0,C 180,E1 -22026.375,E2 -22026.375} C_VEL
LIN {X 0,Y 266.611,Z 1059.755,A -85,B 0,C 180,E1 -22030.957,E2 -22030.957} C_VEL
LIN {X 0,Y 264.694,Z 1065.063,A -85,B 0,C 180,E1 -22036.455,E2 -22036.455} C_VEL
LIN {X 0,Y 264.076,Z 1067.983,A -85,B 0,C 180,E1 -22040.849,E2 -22040.849} C_VEL
LIN {X 0,Y 263.973,Z 1069.66,A -85,B 0,C 180,E1 -22044.784,E2 -22044.784} C_VEL
LIN {X 0,Y 263.999,Z 1070.425,A -85,B 0,C 180,E1 -22048.698,E2 -22048.698} C_VEL
LIN {X 0,Y 263.988,Z 1070.256,A -85,B 0,C 180,E1 -22052.822,E2 -22052.822} C_VEL
LIN {X 0,Y 264.001,Z 1068.785,A -85,B 0,C 180,E1 -22057.617,E2 -22057.617} C_VEL
LIN {X 0,Y 264.475,Z 1065.86,A -85,B 0,C 180,E1 -22062.445,E2 -22062.445} C_VEL
LIN {X 0,Y 265.75,Z 1061.842,A -85,B 0,C 180,E1 -22067.066,E2 -22067.066} C_VEL
LIN {X 0,Y 268.774,Z 1055.118,A -85,B 0,C 180,E1 -22072.689,E2 -22072.689} C_VEL
LIN {X 0,Y 272.709,Z 1047.987,A -85,B 0,C 180,E1 -22077.278,E2 -22077.278} C_VEL
LIN {X 0,Y 279.098,Z 1037.723,A -85,B 0,C 180,E1 -22082.506,E2 -22082.506} C_VEL
LIN {X 0,Y 285.593,Z 1027.883,A -85,B 0,C 180,E1 -22086.526,E2 -22086.526} C_VEL
LIN {X 0,Y 294.132,Z 1015.311,A -85,B 0,C 180,E1 -22090.745,E2 -22090.745} C_VEL
LIN {X 0,Y 302.631,Z 1002.642,A -85,B 0,C 180,E1 -22094.198,E2 -22094.198} C_VEL
LIN {X 0,Y 312.664,Z 987.539,A -85,B 0,C 180,E1 -22097.623,E2 -22097.623} C_VEL
LIN {X 0,Y 323.114,Z 970.828,A -85,B 0,C 180,E1 -22100.681,E2 -22100.681} C_VEL
LIN {X 0,Y 333.509,Z 953.466,A -85,B 0,C 180,E1 -22103.32,E2 -22103.32} C_VEL
LIN {X 0,Y 343.925,Z 934.438,A -85,B 0,C 180,E1 -22105.666,E2 -22105.666} C_VEL
LIN {X 0,Y 353.843,Z 914.962,A -85,B 0,C 180,E1 -22107.662,E2 -22107.662} C_VEL
LIN {X 0,Y 363.336,Z 894.076,A -85,B 0,C 180,E1 -22109.395,E2 -22109.395} C_VEL
LIN {X 0,Y 371.343,Z 874.593,A -85,B 0,C 180,E1 -22110.74,E2 -22110.74} C_VEL
LIN {X 0,Y 379.74,Z 851.133,A -85,B 0,C 180,E1 -22112.051,E2 -22112.051} C_VEL
LIN {X 0,Y 385.909,Z 831.202,A -85,B 0,C 180,E1 -22112.949,E2 -22112.949} C_VEL
LIN {X 0,Y 392.484,Z 805.798,A -85,B 0,C 180,E1 -22113.852,E2 -22113.852} C_VEL
LIN {X 0,Y 396.93,Z 784.071,A -85,B 0,C 180,E1 -22114.44,E2 -22114.44} C_VEL
LIN {X 0,Y 400.768,Z 758.49,A -85,B 0,C 180,E1 -22114.981,E2 -22114.981} C_VEL
LIN {X 0,Y 407.236,Z 683.861,A -85,B 0,C 180,E1 -22116.203,E2 -22116.203} C_VEL
LIN {X 0,Y 417.786,Z 558.474,A -85,B 0,C 180,E1 -22118.225,E2 -22118.225} C_VEL
LIN {X 0,Y 412.702,Z 547.843,A -85,B 0,C 180,E1 -22120.578,E2 -22120.578} C_VEL
LIN {X 0,Y 408.069,Z 538.803,A -85,B 0,C 180,E1 -22123.01,E2 -22123.01} C_VEL
LIN {X 0,Y 403.547,Z 531.446,A -85,B 0,C 180,E1 -22125.727,E2 -22125.727} C_VEL
LIN {X 0,Y 400.615,Z 526.826,A -85,B 0,C 180,E1 -22127.825,E2 -22127.825} C_VEL
LIN {X 0,Y 398.223,Z 522.968,A -85,B 0,C 180,E1 -22129.877,E2 -22129.877} C_VEL
LIN {X 0,Y 395.32,Z 518.27,A -85,B 0,C 180,E1 -22133.173,E2 -22133.173} C_VEL
LIN {X 0,Y 392.974,Z 513.128,A -85,B 0,C 180,E1 -22140.292,E2 -22140.292} C_VEL
LIN {X 0,Y 395.706,Z 518.88,A -85,B 0,C 180,E1 -22147.769,E2 -22147.769} C_VEL
LIN {X 0,Y 398.939,Z 524.131,A -85,B 0,C 180,E1 -22151.201,E2 -22151.201} C_VEL
LIN {X 0,Y 402.153,Z 529.2,A -85,B 0,C 180,E1 -22153.736,E2 -22153.736} C_VEL
LIN {X 0,Y 405.428,Z 534.533,A -85,B 0,C 180,E1 -22155.888,E2 -22155.888} C_VEL
LIN {X 0,Y 410.075,Z 542.205,A -85,B 0,C 180,E1 -22158.481,E2 -22158.481} C_VEL
LIN {X 0,Y 415.899,Z 552.216,A -85,B 0,C 180,E1 -22161.25,E2 -22161.25} C_VEL
LIN {X 0,Y 417.93,Z 556.297,A -85,B 0,C 180,E1 -22162.147,E2 -22162.147} C_VEL
LIN {X 0,Y 401.564,Z 747.417,A -85,B 0,C 180,E1 -22165.21,E2 -22165.21} C_VEL
LIN {X 0,Y 397.773,Z 773.903,A -85,B 0,C 180,E1 -22165.779,E2 -22165.779} C_VEL
LIN {X 0,Y 393.722,Z 794.499,A -85,B 0,C 180,E1 -22166.367,E2 -22166.367} C_VEL
LIN {X 0,Y 387.748,Z 818.868,A -85,B 0,C 180,E1 -22167.259,E2 -22167.259} C_VEL
LIN {X 0,Y 381.377,Z 840.085,A -85,B 0,C 180,E1 -22168.247,E2 -22168.247} C_VEL
LIN {X 0,Y 373.967,Z 861.636,A -85,B 0,C 180,E1 -22169.47,E2 -22169.47} C_VEL
LIN {X 0,Y 365.277,Z 883.119,A -85,B 0,C 180,E1 -22170.972,E2 -22170.972} C_VEL
LIN {X 0,Y 356.323,Z 903.143,A -85,B 0,C 180,E1 -22172.665,E2 -22172.665} C_VEL
LIN {X 0,Y 346.501,Z 922.638,A -85,B 0,C 180,E1 -22174.673,E2 -22174.673} C_VEL
LIN {X 0,Y 337.421,Z 939.282,A -85,B 0,C 180,E1 -22176.719,E2 -22176.719} C_VEL
LIN {X 0,Y 326.438,Z 957.824,A -85,B 0,C 180,E1 -22179.477,E2 -22179.477} C_VEL
LIN {X 0,Y 317.023,Z 972.724,A -85,B 0,C 180,E1 -22182.168,E2 -22182.168} C_VEL
LIN {X 0,Y 306.347,Z 988.779,A -85,B 0,C 180,E1 -22185.695,E2 -22185.695} C_VEL
LIN {X 0,Y 298.085,Z 1000.718,A -85,B 0,C 180,E1 -22188.894,E2 -22188.894} C_VEL
LIN {X 0,Y 289.194,Z 1013.441,A -85,B 0,C 180,E1 -22193.015,E2 -22193.015} C_VEL
LIN {X 0,Y 281.873,Z 1023.819,A -85,B 0,C 180,E1 -22197.216,E2 -22197.216} C_VEL
LIN {X 0,Y 275.581,Z 1033.195,A -85,B 0,C 180,E1 -22201.857,E2 -22201.857} C_VEL
LIN {X 0,Y 270.727,Z 1040.798,A -85,B 0,C 180,E1 -22206.722,E2 -22206.722} C_VEL
LIN {X 0,Y 267.482,Z 1046.677,A -85,B 0,C 180,E1 -22211.474,E2 -22211.474} C_VEL
LIN {X 0,Y 265.319,Z 1051.405,A -85,B 0,C 180,E1 -22216.71,E2 -22216.71} C_VEL
LIN {X 0,Y 264.419,Z 1054.124,A -85,B 0,C 180,E1 -22221.081,E2 -22221.081} C_VEL
LIN {X 0,Y 264.09,Z 1055.73,A -85,B 0,C 180,E1 -22225.222,E2 -22225.222} C_VEL
LIN {X 0,Y 264.016,Z 1056.461,A -85,B 0,C 180,E1 -22230,E2 -22230} C_VEL
LIN {X 0,Y 264.089,Z 1055.769,A -85,B 0,C 180,E1 -22234.778,E2 -22234.778} C_VEL
LIN {X 0,Y 264.439,Z 1054.079,A -85,B 0,C 180,E1 -22239.138,E2 -22239.138} C_VEL
LIN {X 0,Y 265.427,Z 1051.185,A -85,B 0,C 180,E1 -22243.729,E2 -22243.729} C_VEL
LIN {X 0,Y 267.803,Z 1046.074,A -85,B 0,C 180,E1 -22249.182,E2 -22249.182} C_VEL
LIN {X 0,Y 271.026,Z 1040.375,A -85,B 0,C 180,E1 -22253.712,E2 -22253.712} C_VEL
LIN {X 0,Y 276.37,Z 1032.024,A -85,B 0,C 180,E1 -22258.89,E2 -22258.89} C_VEL
LIN {X 0,Y 282.188,Z 1023.456,A -85,B 0,C 180,E1 -22263.071,E2 -22263.071} C_VEL
LIN {X 0,Y 289.826,Z 1012.696,A -85,B 0,C 180,E1 -22267.387,E2 -22267.387} C_VEL
LIN {X 0,Y 298.606,Z 1000.114,A -85,B 0,C 180,E1 -22271.403,E2 -22271.403} C_VEL
LIN {X 0,Y 308.152,Z 986.383,A -85,B 0,C 180,E1 -22275.021,E2 -22275.021} C_VEL
LIN {X 0,Y 317.939,Z 971.5,A -85,B 0,C 180,E1 -22278.189,E2 -22278.189} C_VEL
LIN {X 0,Y 327.432,Z 956.476,A -85,B 0,C 180,E1 -22280.864,E2 -22280.864} C_VEL
LIN {X 0,Y 338.173,Z 938.209,A -85,B 0,C 180,E1 -22283.537,E2 -22283.537} C_VEL
LIN {X 0,Y 347.299,Z 921.461,A -85,B 0,C 180,E1 -22285.573,E2 -22285.573} C_VEL
LIN {X 0,Y 357.819,Z 900.257,A -85,B 0,C 180,E1 -22287.705,E2 -22287.705} C_VEL
LIN {X 0,Y 365.984,Z 881.905,A -85,B 0,C 180,E1 -22289.231,E2 -22289.231} C_VEL
LIN {X 0,Y 374.774,Z 859.886,A -85,B 0,C 180,E1 -22290.743,E2 -22290.743} C_VEL
LIN {X 0,Y 381.929,Z 838.972,A -85,B 0,C 180,E1 -22291.917,E2 -22291.917} C_VEL
LIN {X 0,Y 388.736,Z 816.089,A -85,B 0,C 180,E1 -22292.965,E2 -22292.965} C_VEL
LIN {X 0,Y 394.327,Z 792.621,A -85,B 0,C 180,E1 -22293.798,E2 -22293.798} C_VEL
LIN {X 0,Y 398.729,Z 769.763,A -85,B 0,C 180,E1 -22294.431,E2 -22294.431} C_VEL
LIN {X 0,Y 402.018,Z 745.045,A -85,B 0,C 180,E1 -22294.937,E2 -22294.937} C_VEL
LIN {X 0,Y 412.944,Z 617.12,A -85,B 0,C 180,E1 -22296.995,E2 -22296.995} C_VEL
LIN {X 0,Y 413.211,Z 609.563,A -85,B 0,C 180,E1 -22297.24,E2 -22297.24} C_VEL
LIN {X 0,Y 412.559,Z 589.904,A -85,B 0,C 180,E1 -22298.356,E2 -22298.356} C_VEL
LIN {X 0,Y 412.85,Z 583.407,A -85,B 0,C 180,E1 -22298.557,E2 -22298.557} C_VEL
LIN {X 0,Y 414.782,Z 560.925,A -85,B 0,C 180,E1 -22298.925,E2 -22298.925} C_VEL
LIN {X 0,Y 409.321,Z 551.112,A -85,B 0,C 180,E1 -22301.558,E2 -22301.558} C_VEL
LIN {X 0,Y 404.247,Z 542.501,A -85,B 0,C 180,E1 -22304.433,E2 -22304.433} C_VEL
LIN {X 0,Y 401.139,Z 537.359,A -85,B 0,C 180,E1 -22306.523,E2 -22306.523} C_VEL
LIN {X 0,Y 399.214,Z 534.347,A -85,B 0,C 180,E1 -22308.001,E2 -22308.001} C_VEL
LIN {X 0,Y 397.021,Z 530.697,A -85,B 0,C 180,E1 -22309.993,E2 -22309.993} C_VEL
LIN {X 0,Y 394.398,Z 526.264,A -85,B 0,C 180,E1 -22313.157,E2 -22313.157} C_VEL
LIN {X 0,Y 392.24,Z 522.044,A -85,B 0,C 180,E1 -22319.854,E2 -22319.854} C_VEL
LIN {X 0,Y 394.731,Z 526.749,A -85,B 0,C 180,E1 -22326.984,E2 -22326.984} C_VEL
LIN {X 0,Y 397.885,Z 532.026,A -85,B 0,C 180,E1 -22330.498,E2 -22330.498} C_VEL
LIN {X 0,Y 400.71,Z 536.665,A -85,B 0,C 180,E1 -22332.831,E2 -22332.831} C_VEL
LIN {X 0,Y 404.191,Z 542.412,A -85,B 0,C 180,E1 -22335.202,E2 -22335.202} C_VEL
LIN {X 0,Y 407.582,Z 548.306,A -85,B 0,C 180,E1 -22337.194,E2 -22337.194} C_VEL
LIN {X 0,Y 412.895,Z 559.27,A -85,B 0,C 180,E1 -22339.966,E2 -22339.966} C_VEL
LIN {X 0,Y 414.709,Z 563.568,A -85,B 0,C 180,E1 -22340.843,E2 -22340.843} C_VEL
LIN {X 0,Y 397.844,Z 756.431,A -85,B 0,C 180,E1 -22343.924,E2 -22343.924} C_VEL
LIN {X 0,Y 393.879,Z 783.115,A -85,B 0,C 180,E1 -22344.473,E2 -22344.473} C_VEL
LIN {X 0,Y 389.445,Z 804.551,A -85,B 0,C 180,E1 -22345.04,E2 -22345.04} C_VEL
LIN {X 0,Y 382.933,Z 829.586,A -85,B 0,C 180,E1 -22345.903,E2 -22345.903} C_VEL
LIN {X 0,Y 376.807,Z 849.12,A -85,B 0,C 180,E1 -22346.756,E2 -22346.756} C_VEL
LIN {X 0,Y 368.947,Z 871.117,A -85,B 0,C 180,E1 -22347.933,E2 -22347.933} C_VEL
LIN {X 0,Y 359.821,Z 893.009,A -85,B 0,C 180,E1 -22349.405,E2 -22349.405} C_VEL
LIN {X 0,Y 350.262,Z 913.646,A -85,B 0,C 180,E1 -22351.084,E2 -22351.084} C_VEL
LIN {X 0,Y 340.039,Z 933.296,A -85,B 0,C 180,E1 -22353.065,E2 -22353.065} C_VEL
LIN {X 0,Y 330.262,Z 950.701,A -85,B 0,C 180,E1 -22355.17,E2 -22355.17} C_VEL
LIN {X 0,Y 318.985,Z 969.199,A -85,B 0,C 180,E1 -22357.907,E2 -22357.907} C_VEL
LIN {X 0,Y 309.36,Z 984.082,A -85,B 0,C 180,E1 -22360.575,E2 -22360.575} C_VEL
LIN {X 0,Y 298.264,Z 1000.43,A -85,B 0,C 180,E1 -22364.159,E2 -22364.159} C_VEL
LIN {X 0,Y 289.24,Z 1013.276,A -85,B 0,C 180,E1 -22367.615,E2 -22367.615} C_VEL
LIN {X 0,Y 279.352,Z 1027.227,A -85,B 0,C 180,E1 -22372.261,E2 -22372.261} C_VEL
LIN {X 0,Y 272.46,Z 1037.115,A -85,B 0,C 180,E1 -22376.348,E2 -22376.348} C_VEL
LIN {X 0,Y 265.624,Z 1047.469,A -85,B 0,C 180,E1 -22381.686,E2 -22381.686} C_VEL
LIN {X 0,Y 261.413,Z 1054.543,A -85,B 0,C 180,E1 -22386.32,E2 -22386.32} C_VEL
LIN {X 0,Y 258.218,Z 1061.019,A -85,B 0,C 180,E1 -22391.72,E2 -22391.72} C_VEL
LIN {X 0,Y 256.631,Z 1065.341,A -85,B 0,C 180,E1 -22396.71,E2 -22396.71} C_VEL
LIN {X 0,Y 256.056,Z 1068.12,A -85,B 0,C 180,E1 -22401.24,E2 -22401.24} C_VEL
LIN {X 0,Y 255.976,Z 1069.935,A -85,B 0,C 180,E1 -22406.192,E2 -22406.192} C_VEL
LIN {X 0,Y 256.007,Z 1070.278,A -85,B 0,C 180,E1 -22410.671,E2 -22410.671} C_VEL
LIN {X 0,Y 255.975,Z 1069.531,A -85,B 0,C 180,E1 -22415.071,E2 -22415.071} C_VEL
LIN {X 0,Y 256.079,Z 1067.866,A -85,B 0,C 180,E1 -22419.212,E2 -22419.212} C_VEL
LIN {X 0,Y 256.728,Z 1064.984,A -85,B 0,C 180,E1 -22423.744,E2 -22423.744} C_VEL
LIN {X 0,Y 258.778,Z 1059.682,A -85,B 0,C 180,E1 -22429.474,E2 -22429.474} C_VEL
LIN {X 0,Y 261.751,Z 1053.869,A -85,B 0,C 180,E1 -22434.126,E2 -22434.126} C_VEL
LIN {X 0,Y 266.584,Z 1045.961,A -85,B 0,C 180,E1 -22439.183,E2 -22439.183} C_VEL
LIN {X 0,Y 273.085,Z 1036.101,A -85,B 0,C 180,E1 -22444.07,E2 -22444.07} C_VEL
LIN {X 0,Y 280.871,Z 1025.046,A -85,B 0,C 180,E1 -22448.535,E2 -22448.535} C_VEL
LIN {X 0,Y 289.676,Z 1012.514,A -85,B 0,C 180,E1 -22452.574,E2 -22452.574} C_VEL
LIN {X 0,Y 298.75,Z 999.584,A -85,B 0,C 180,E1 -22456.02,E2 -22456.02} C_VEL
LIN {X 0,Y 309.722,Z 983.325,A -85,B 0,C 180,E1 -22459.541,E2 -22459.541} C_VEL
LIN {X 0,Y 319.137,Z 968.736,A -85,B 0,C 180,E1 -22462.142,E2 -22462.142} C_VEL
LIN {X 0,Y 330.875,Z 949.349,A -85,B 0,C 180,E1 -22464.979,E2 -22464.979} C_VEL
LIN {X 0,Y 340.349,Z 932.418,A -85,B 0,C 180,E1 -22467.008,E2 -22467.008} C_VEL
LIN {X 0,Y 350.928,Z 911.838,A -85,B 0,C 180,E1 -22469.051,E2 -22469.051} C_VEL
LIN {X 0,Y 359.794,Z 892.644,A -85,B 0,C 180,E1 -22470.602,E2 -22470.602} C_VEL
LIN {X 0,Y 368.919,Z 870.67,A -85,B 0,C 180,E1 -22472.075,E2 -22472.075} C_VEL
LIN {X 0,Y 376.666,Z 848.953,A -85,B 0,C 180,E1 -22473.235,E2 -22473.235} C_VEL
LIN {X 0,Y 383.295,Z 827.708,A -85,B 0,C 180,E1 -22474.156,E2 -22474.156} C_VEL
LIN {X 0,Y 389.414,Z 803.769,A -85,B 0,C 180,E1 -22474.967,E2 -22474.967} C_VEL
LIN {X 0,Y 393.827,Z 782.275,A -85,B 0,C 180,E1 -22475.532,E2 -22475.532} C_VEL
LIN {X 0,Y 397.72,Z 755.572,A -85,B 0,C 180,E1 -22476.077,E2 -22476.077} C_VEL
LIN {X 0,Y 414.506,Z 563.105,A -85,B 0,C 180,E1 -22479.157,E2 -22479.157} C_VEL
LIN {X 0,Y 410.112,Z 553.809,A -85,B 0,C 180,E1 -22481.3,E2 -22481.3} C_VEL
LIN {X 0,Y 406.206,Z 545.961,A -85,B 0,C 180,E1 -22483.446,E2 -22483.446} C_VEL
LIN {X 0,Y 401.823,Z 538.688,A -85,B 0,C 180,E1 -22486.179,E2 -22486.179} C_VEL
LIN {X 0,Y 399.177,Z 534.386,A -85,B 0,C 180,E1 -22488.147,E2 -22488.147} C_VEL
LIN {X 0,Y 396.937,Z 530.68,A -85,B 0,C 180,E1 -22490.137,E2 -22490.137} C_VEL
LIN {X 0,Y 394.237,Z 526.155,A -85,B 0,C 180,E1 -22493.3,E2 -22493.3} C_VEL
LIN {X 0,Y 391.992,Z 521.119,A -85,B 0,C 180,E1 -22500.292,E2 -22500.292} C_VEL
LIN {X 0,Y 394.56,Z 526.698,A -85,B 0,C 180,E1 -22507.572,E2 -22507.572} C_VEL
LIN {X 0,Y 397.634,Z 531.828,A -85,B 0,C 180,E1 -22510.944,E2 -22510.944} C_VEL
LIN {X 0,Y 400.769,Z 536.914,A -85,B 0,C 180,E1 -22513.49,E2 -22513.49} C_VEL
LIN {X 0,Y 404.895,Z 543.669,A -85,B 0,C 180,E1 -22516.204,E2 -22516.204} C_VEL
LIN {X 0,Y 410.187,Z 552.886,A -85,B 0,C 180,E1 -22519.102,E2 -22519.102} C_VEL
LIN {X 0,Y 414.591,Z 560.948,A -85,B 0,C 180,E1 -22521.192,E2 -22521.192} C_VEL
LIN {X 0,Y 398.222,Z 747.653,A -85,B 0,C 180,E1 -22524.168,E2 -22524.168} C_VEL
LIN {X 0,Y 394.344,Z 774.197,A -85,B 0,C 180,E1 -22524.733,E2 -22524.733} C_VEL
LIN {X 0,Y 390.184,Z 794.919,A -85,B 0,C 180,E1 -22525.319,E2 -22525.319} C_VEL
LIN {X 0,Y 384.106,Z 819.189,A -85,B 0,C 180,E1 -22526.198,E2 -22526.198} C_VEL
LIN {X 0,Y 377.636,Z 840.307,A -85,B 0,C 180,E1 -22527.171,E2 -22527.171} C_VEL
LIN {X 0,Y 369.619,Z 862.997,A -85,B 0,C 180,E1 -22528.456,E2 -22528.456} C_VEL
LIN {X 0,Y 361.007,Z 883.749,A -85,B 0,C 180,E1 -22529.904,E2 -22529.904} C_VEL
LIN {X 0,Y 351.676,Z 904.094,A -85,B 0,C 180,E1 -22531.621,E2 -22531.621} C_VEL
LIN {X 0,Y 341.615,Z 923.463,A -85,B 0,C 180,E1 -22533.622,E2 -22533.622} C_VEL
LIN {X 0,Y 331.676,Z 941.155,A -85,B 0,C 180,E1 -22535.812,E2 -22535.812} C_VEL
LIN {X 0,Y 320.716,Z 958.962,A -85,B 0,C 180,E1 -22538.507,E2 -22538.507} C_VEL
LIN {X 0,Y 310.971,Z 973.884,A -85,B 0,C 180,E1 -22541.236,E2 -22541.236} C_VEL
LIN {X 0,Y 300.029,Z 989.693,A -85,B 0,C 180,E1 -22544.777,E2 -22544.777} C_VEL
LIN {X 0,Y 291.495,Z 1001.566,A -85,B 0,C 180,E1 -22548.019,E2 -22548.019} C_VEL
LIN {X 0,Y 281.891,Z 1014.676,A -85,B 0,C 180,E1 -22552.404,E2 -22552.404} C_VEL
LIN {X 0,Y 274.734,Z 1024.405,A -85,B 0,C 180,E1 -22556.454,E2 -22556.454} C_VEL
LIN {X 0,Y 268.111,Z 1033.766,A -85,B 0,C 180,E1 -22561.244,E2 -22561.244} C_VEL
LIN {X 0,Y 263.039,Z 1041.315,A -85,B 0,C 180,E1 -22566.238,E2 -22566.238} C_VEL
LIN {X 0,Y 259.397,Z 1047.625,A -85,B 0,C 180,E1 -22571.574,E2 -22571.574} C_VEL
LIN {X 0,Y 257.305,Z 1051.932,A -85,B 0,C 180,E1 -22576.746,E2 -22576.746} C_VEL
LIN {X 0,Y 256.399,Z 1054.56,A -85,B 0,C 180,E1 -22581.252,E2 -22581.252} C_VEL
LIN {X 0,Y 256.06,Z 1056.276,A -85,B 0,C 180,E1 -22586.194,E2 -22586.194} C_VEL
LIN {X 0,Y 256.017,Z 1056.576,A -85,B 0,C 180,E1 -22591.119,E2 -22591.119} C_VEL
LIN {X 0,Y 256.117,Z 1055.84,A -85,B 0,C 180,E1 -22595.416,E2 -22595.416} C_VEL
LIN {X 0,Y 256.524,Z 1054.184,A -85,B 0,C 180,E1 -22599.649,E2 -22599.649} C_VEL
LIN {X 0,Y 257.789,Z 1050.936,A -85,B 0,C 180,E1 -22604.833,E2 -22604.833} C_VEL
LIN {X 0,Y 260.385,Z 1045.794,A -85,B 0,C 180,E1 -22610.219,E2 -22610.219} C_VEL
LIN {X 0,Y 264.147,Z 1039.703,A -85,B 0,C 180,E1 -22615.085,E2 -22615.085} C_VEL
LIN {X 0,Y 270.02,Z 1031.055,A -85,B 0,C 180,E1 -22620.366,E2 -22620.366} C_VEL
LIN {X 0,Y 276.337,Z 1022.32,A -85,B 0,C 180,E1 -22624.617,E2 -22624.617} C_VEL
LIN {X 0,Y 285.339,Z 1010.095,A -85,B 0,C 180,E1 -22629.366,E2 -22629.366} C_VEL
LIN {X 0,Y 293.702,Z 998.682,A -85,B 0,C 180,E1 -22632.949,E2 -22632.949} C_VEL
LIN {X 0,Y 304.465,Z 983.567,A -85,B 0,C 180,E1 -22636.809,E2 -22636.809} C_VEL
LIN {X 0,Y 314.017,Z 969.521,A -85,B 0,C 180,E1 -22639.73,E2 -22639.73} C_VEL
LIN {X 0,Y 325.351,Z 951.871,A -85,B 0,C 180,E1 -22642.748,E2 -22642.748} C_VEL
LIN {X 0,Y 334.667,Z 936.22,A -85,B 0,C 180,E1 -22644.949,E2 -22644.949} C_VEL
LIN {X 0,Y 345.107,Z 917.417,A -85,B 0,C 180,E1 -22647.164,E2 -22647.164} C_VEL
LIN {X 0,Y 354.588,Z 898.277,A -85,B 0,C 180,E1 -22649.008,E2 -22649.008} C_VEL
LIN {X 0,Y 362.992,Z 879.693,A -85,B 0,C 180,E1 -22650.511,E2 -22650.511} C_VEL
LIN {X 0,Y 371.971,Z 857.138,A -85,B 0,C 180,E1 -22652.004,E2 -22652.004} C_VEL
LIN {X 0,Y 378.548,Z 838.149,A -85,B 0,C 180,E1 -22653.044,E2 -22653.044} C_VEL
LIN {X 0,Y 385.674,Z 814.216,A -85,B 0,C 180,E1 -22654.109,E2 -22654.109} C_VEL
LIN {X 0,Y 391.062,Z 791.856,A -85,B 0,C 180,E1 -22654.883,E2 -22654.883} C_VEL
LIN {X 0,Y 395.678,Z 767.914,A -85,B 0,C 180,E1 -22655.527,E2 -22655.527} C_VEL
LIN {X 0,Y 398.84,Z 743.846,A -85,B 0,C 180,E1 -22656.003,E2 -22656.003} C_VEL
LIN {X 0,Y 412.85,Z 583.407,A -85,B 0,C 180,E1 -22658.557,E2 -22658.557} C_VEL
LIN {X 0,Y 413.029,Z 577.423,A -85,B 0,C 180,E1 -22658.775,E2 -22658.775} C_VEL
LIN {X 0,Y 412.526,Z 571.34,A -85,B 0,C 180,E1 -22659.25,E2 -22659.25} C_VEL
LIN {X 0,Y 411.434,Z 566.285,A -85,B 0,C 180,E1 -22659.911,E2 -22659.911} C_VEL
LIN {X 0,Y 410.414,Z 563.729,A -85,B 0,C 180,E1 -22660.439,E2 -22660.439} C_VEL
LIN {X 0,Y 405.192,Z 554.364,A -85,B 0,C 180,E1 -22663.219,E2 -22663.219} C_VEL
LIN {X 0,Y 400.736,Z 546.624,A -85,B 0,C 180,E1 -22666.067,E2 -22666.067} C_VEL
LIN {X 0,Y 398.143,Z 542.411,A -85,B 0,C 180,E1 -22668.042,E2 -22668.042} C_VEL
LIN {X 0,Y 395.751,Z 538.411,A -85,B 0,C 180,E1 -22670.254,E2 -22670.254} C_VEL
LIN {X 0,Y 393.322,Z 534.148,A -85,B 0,C 180,E1 -22673.284,E2 -22673.284} C_VEL
LIN {X 0,Y 391.264,Z 529.992,A -85,B 0,C 180,E1 -22679.854,E2 -22679.854} C_VEL
LIN {X 0,Y 393.595,Z 534.56,A -85,B 0,C 180,E1 -22686.784,E2 -22686.784} C_VEL
LIN {X 0,Y 396.591,Z 539.718,A -85,B 0,C 180,E1 -22690.239,E2 -22690.239} C_VEL
LIN {X 0,Y 399.432,Z 544.546,A -85,B 0,C 180,E1 -22692.653,E2 -22692.653} C_VEL
LIN {X 0,Y 402.86,Z 550.312,A -85,B 0,C 180,E1 -22695.033,E2 -22695.033} C_VEL
LIN {X 0,Y 405.827,Z 555.705,A -85,B 0,C 180,E1 -22696.828,E2 -22696.828} C_VEL
LIN {X 0,Y 410.806,Z 566.292,A -85,B 0,C 180,E1 -22699.516,E2 -22699.516} C_VEL
LIN {X 0,Y 411.481,Z 568.232,A -85,B 0,C 180,E1 -22699.874,E2 -22699.874} C_VEL
LIN {X 0,Y 394.656,Z 756.238,A -85,B 0,C 180,E1 -22702.858,E2 -22702.858} C_VEL
LIN {X 0,Y 390.62,Z 782.913,A -85,B 0,C 180,E1 -22703.4,E2 -22703.4} C_VEL
LIN {X 0,Y 386.106,Z 804.365,A -85,B 0,C 180,E1 -22703.959,E2 -22703.959} C_VEL
LIN {X 0,Y 379.481,Z 829.379,A -85,B 0,C 180,E1 -22704.808,E2 -22704.808} C_VEL
LIN {X 0,Y 373.086,Z 849.358,A -85,B 0,C 180,E1 -22705.669,E2 -22705.669} C_VEL
LIN {X 0,Y 364.842,Z 871.848,A -85,B 0,C 180,E1 -22706.866,E2 -22706.866} C_VEL
LIN {X 0,Y 356.03,Z 892.505,A -85,B 0,C 180,E1 -22708.243,E2 -22708.243} C_VEL
LIN {X 0,Y 346.59,Z 912.456,A -85,B 0,C 180,E1 -22709.843,E2 -22709.843} C_VEL
LIN {X 0,Y 335.986,Z 932.469,A -85,B 0,C 180,E1 -22711.827,E2 -22711.827} C_VEL
LIN {X 0,Y 326.257,Z 949.367,A -85,B 0,C 180,E1 -22713.845,E2 -22713.845} C_VEL
LIN {X 0,Y 314.169,Z 968.709,A -85,B 0,C 180,E1 -22716.676,E2 -22716.676} C_VEL
LIN {X 0,Y 304.051,Z 983.864,A -85,B 0,C 180,E1 -22719.393,E2 -22719.393} C_VEL
LIN {X 0,Y 292.554,Z 1000.211,A -85,B 0,C 180,E1 -22722.995,E2 -22722.995} C_VEL
LIN {X 0,Y 283.174,Z 1013.057,A -85,B 0,C 180,E1 -22726.485,E2 -22726.485} C_VEL
LIN {X 0,Y 272.836,Z 1027.007,A -85,B 0,C 180,E1 -22731.194,E2 -22731.194} C_VEL
LIN {X 0,Y 265.597,Z 1036.895,A -85,B 0,C 180,E1 -22735.356,E2 -22735.356} C_VEL
LIN {X 0,Y 258.371,Z 1047.249,A -85,B 0,C 180,E1 -22740.816,E2 -22740.816} C_VEL
LIN {X 0,Y 253.881,Z 1054.323,A -85,B 0,C 180,E1 -22745.573,E2 -22745.573} C_VEL
LIN {X 0,Y 250.444,Z 1060.801,A -85,B 0,C 180,E1 -22751.132,E2 -22751.132} C_VEL
LIN {X 0,Y 248.714,Z 1065.124,A -85,B 0,C 180,E1 -22756.279,E2 -22756.279} C_VEL
LIN {X 0,Y 248.07,Z 1067.905,A -85,B 0,C 180,E1 -22760.956,E2 -22760.956} C_VEL
LIN {X 0,Y 247.976,Z 1069.653,A -85,B 0,C 180,E1 -22765.838,E2 -22765.838} C_VEL
LIN {X 0,Y 248.011,Z 1070.087,A -85,B 0,C 180,E1 -22770.462,E2 -22770.462} C_VEL
LIN {X 0,Y 247.977,Z 1069.36,A -85,B 0,C 180,E1 -22775.089,E2 -22775.089} C_VEL
LIN {X 0,Y 248.098,Z 1067.65,A -85,B 0,C 180,E1 -22779.511,E2 -22779.511} C_VEL
LIN {X 0,Y 248.818,Z 1064.766,A -85,B 0,C 180,E1 -22784.189,E2 -22784.189} C_VEL
LIN {X 0,Y 251.017,Z 1059.535,A -85,B 0,C 180,E1 -22790.033,E2 -22790.033} C_VEL
LIN {X 0,Y 254.426,Z 1053.338,A -85,B 0,C 180,E1 -22795.115,E2 -22795.115} C_VEL
LIN {X 0,Y 259.905,Z 1044.931,A -85,B 0,C 180,E1 -22800.519,E2 -22800.519} C_VEL
LIN {X 0,Y 266.59,Z 1035.412,A -85,B 0,C 180,E1 -22805.282,E2 -22805.282} C_VEL
LIN {X 0,Y 275.014,Z 1024.031,A -85,B 0,C 180,E1 -22809.901,E2 -22809.901} C_VEL
LIN {X 0,Y 284.098,Z 1011.648,A -85,B 0,C 180,E1 -22813.895,E2 -22813.895} C_VEL
LIN {X 0,Y 294.112,Z 997.943,A -85,B 0,C 180,E1 -22817.538,E2 -22817.538} C_VEL
LIN {X 0,Y 304.606,Z 982.834,A -85,B 0,C 180,E1 -22820.776,E2 -22820.776} C_VEL
LIN {X 0,Y 314.765,Z 967.579,A -85,B 0,C 180,E1 -22823.483,E2 -22823.483} C_VEL
LIN {X 0,Y 326.564,Z 948.567,A -85,B 0,C 180,E1 -22826.231,E2 -22826.231} C_VEL
LIN {X 0,Y 336.317,Z 931.563,A -85,B 0,C 180,E1 -22828.249,E2 -22828.249} C_VEL
LIN {X 0,Y 347.583,Z 910.009,A -85,B 0,C 180,E1 -22830.344,E2 -22830.344} C_VEL
LIN {X 0,Y 356.241,Z 891.607,A -85,B 0,C 180,E1 -22831.803,E2 -22831.803} C_VEL
LIN {X 0,Y 365.524,Z 869.552,A -85,B 0,C 180,E1 -22833.251,E2 -22833.251} C_VEL
LIN {X 0,Y 373.152,Z 848.559,A -85,B 0,C 180,E1 -22834.352,E2 -22834.352} C_VEL
LIN {X 0,Y 380.204,Z 826.325,A -85,B 0,C 180,E1 -22835.297,E2 -22835.297} C_VEL
LIN {X 0,Y 386.261,Z 802.753,A -85,B 0,C 180,E1 -22836.071,E2 -22836.071} C_VEL
LIN {X 0,Y 390.789,Z 780.9,A -85,B 0,C 180,E1 -22836.632,E2 -22836.632} C_VEL
LIN {X 0,Y 394.577,Z 754.907,A -85,B 0,C 180,E1 -22837.151,E2 -22837.151} C_VEL
LIN {X 0,Y 411.259,Z 567.659,A -85,B 0,C 180,E1 -22840.137,E2 -22840.137} C_VEL
LIN {X 0,Y 406.855,Z 558.132,A -85,B 0,C 180,E1 -22842.442,E2 -22842.442} C_VEL
LIN {X 0,Y 404.077,Z 552.602,A -85,B 0,C 180,E1 -22844.058,E2 -22844.058} C_VEL
LIN {X 0,Y 400.026,Z 545.767,A -85,B 0,C 180,E1 -22846.705,E2 -22846.705} C_VEL
LIN {X 0,Y 397.668,Z 541.813,A -85,B 0,C 180,E1 -22848.543,E2 -22848.543} C_VEL
LIN {X 0,Y 395.658,Z 538.39,A -85,B 0,C 180,E1 -22850.399,E2 -22850.399} C_VEL
LIN {X 0,Y 393.156,Z 534.04,A -85,B 0,C 180,E1 -22853.428,E2 -22853.428} C_VEL
LIN {X 0,Y 391.011,Z 529.109,A -85,B 0,C 180,E1 -22860.293,E2 -22860.293} C_VEL
LIN {X 0,Y 393.466,Z 534.638,A -85,B 0,C 180,E1 -22867.447,E2 -22867.447} C_VEL
LIN {X 0,Y 396.411,Z 539.673,A -85,B 0,C 180,E1 -22870.758,E2 -22870.758} C_VEL
LIN {X 0,Y 399.392,Z 544.627,A -85,B 0,C 180,E1 -22873.243,E2 -22873.243} C_VEL
LIN {X 0,Y 403.376,Z 551.335,A -85,B 0,C 180,E1 -22875.934,E2 -22875.934} C_VEL
LIN {X 0,Y 408.564,Z 560.631,A -85,B 0,C 180,E1 -22878.847,E2 -22878.847} C_VEL
LIN {X 0,Y 411.344,Z 565.861,A -85,B 0,C 180,E1 -22880.226,E2 -22880.226} C_VEL
LIN {X 0,Y 395.013,Z 747.889,A -85,B 0,C 180,E1 -22883.109,E2 -22883.109} C_VEL
LIN {X 0,Y 391.065,Z 774.407,A -85,B 0,C 180,E1 -22883.667,E2 -22883.667} C_VEL
LIN {X 0,Y 386.837,Z 795.084,A -85,B 0,C 180,E1 -22884.243,E2 -22884.243} C_VEL
LIN {X 0,Y 380.599,Z 819.508,A -85,B 0,C 180,E1 -22885.117,E2 -22885.117} C_VEL
LIN {X 0,Y 374.031,Z 840.53,A -85,B 0,C 180,E1 -22886.075,E2 -22886.075} C_VEL
LIN {X 0,Y 366.021,Z 862.798,A -85,B 0,C 180,E1 -22887.319,E2 -22887.319} C_VEL
LIN {X 0,Y 357.065,Z 883.933,A -85,B 0,C 180,E1 -22888.778,E2 -22888.778} C_VEL
LIN {X 0,Y 347.846,Z 903.585,A -85,B 0,C 180,E1 -22890.418,E2 -22890.418} C_VEL
LIN {X 0,Y 337.297,Z 923.486,A -85,B 0,C 180,E1 -22892.45,E2 -22892.45} C_VEL
LIN {X 0,Y 327.3,Z 940.825,A -85,B 0,C 180,E1 -22894.582,E2 -22894.582} C_VEL
LIN {X 0,Y 316.309,Z 958.266,A -85,B 0,C 180,E1 -22897.193,E2 -22897.193} C_VEL
LIN {X 0,Y 306.277,Z 973.167,A -85,B 0,C 180,E1 -22899.898,E2 -22899.898} C_VEL
LIN {X 0,Y 294.546,Z 989.593,A -85,B 0,C 180,E1 -22903.561,E2 -22903.561} C_VEL
LIN {X 0,Y 285.441,Z 1001.788,A -85,B 0,C 180,E1 -22906.916,E2 -22906.916} C_VEL
LIN {X 0,Y 275.421,Z 1014.898,A -85,B 0,C 180,E1 -22911.36,E2 -22911.36} C_VEL
LIN {X 0,Y 267.976,Z 1024.552,A -85,B 0,C 180,E1 -22915.448,E2 -22915.448} C_VEL
LIN {X 0,Y 260.791,Z 1034.179,A -85,B 0,C 180,E1 -22920.498,E2 -22920.498} C_VEL
LIN {X 0,Y 255.565,Z 1041.534,A -85,B 0,C 180,E1 -22925.498,E2 -22925.498} C_VEL
LIN {X 0,Y 251.677,Z 1047.844,A -85,B 0,C 180,E1 -22930.987,E2 -22930.987} C_VEL
LIN {X 0,Y 249.421,Z 1052.148,A -85,B 0,C 180,E1 -22936.319,E2 -22936.319} C_VEL
LIN {X 0,Y 248.441,Z 1054.776,A -85,B 0,C 180,E1 -22940.97,E2 -22940.97} C_VEL
LIN {X 0,Y 248.067,Z 1056.49,A -85,B 0,C 180,E1 -22946.071,E2 -22946.071} C_VEL
LIN {X 0,Y 248.021,Z 1056.794,A -85,B 0,C 180,E1 -22951.115,E2 -22951.115} C_VEL
LIN {X 0,Y 248.127,Z 1056.065,A -85,B 0,C 180,E1 -22955.55,E2 -22955.55} C_VEL
LIN {X 0,Y 248.568,Z 1054.399,A -85,B 0,C 180,E1 -22959.961,E2 -22959.961} C_VEL
LIN {X 0,Y 249.997,Z 1051.059,A -85,B 0,C 180,E1 -22965.44,E2 -22965.44} C_VEL
LIN {X 0,Y 252.737,Z 1046.011,A -85,B 0,C 180,E1 -22970.859,E2 -22970.859} C_VEL
LIN {X 0,Y 256.8,Z 1039.848,A -85,B 0,C 180,E1 -22975.915,E2 -22975.915} C_VEL
LIN {X 0,Y 262.813,Z 1031.479,A -85,B 0,C 180,E1 -22981.16,E2 -22981.16} C_VEL
LIN {X 0,Y 269.254,Z 1022.989,A -85,B 0,C 180,E1 -22985.403,E2 -22985.403} C_VEL
LIN {X 0,Y 278.604,Z 1010.878,A -85,B 0,C 180,E1 -22990.241,E2 -22990.241} C_VEL
LIN {X 0,Y 287.388,Z 999.36,A -85,B 0,C 180,E1 -22993.928,E2 -22993.928} C_VEL
LIN {X 0,Y 298.377,Z 984.546,A -85,B 0,C 180,E1 -22997.782,E2 -22997.782} C_VEL
LIN {X 0,Y 308.443,Z 970.237,A -85,B 0,C 180,E1 -23000.792,E2 -23000.792} C_VEL
LIN {X 0,Y 319.856,Z 953.09,A -85,B 0,C 180,E1 -23003.758,E2 -23003.758} C_VEL
LIN {X 0,Y 330.056,Z 936.434,A -85,B 0,C 180,E1 -23006.106,E2 -23006.106} C_VEL
LIN {X 0,Y 340.825,Z 917.527,A -85,B 0,C 180,E1 -23008.322,E2 -23008.322} C_VEL
LIN {X 0,Y 350.837,Z 897.758,A -85,B 0,C 180,E1 -23010.207,E2 -23010.207} C_VEL
LIN {X 0,Y 360.188,Z 877.48,A -85,B 0,C 180,E1 -23011.81,E2 -23011.81} C_VEL
LIN {X 0,Y 368.646,Z 856.302,A -85,B 0,C 180,E1 -23013.171,E2 -23013.171} C_VEL
LIN {X 0,Y 375.764,Z 836.009,A -85,B 0,C 180,E1 -23014.255,E2 -23014.255} C_VEL
LIN {X 0,Y 383,Z 811.47,A -85,B 0,C 180,E1 -23015.301,E2 -23015.301} C_VEL
LIN {X 0,Y 388.295,Z 789.501,A -85,B 0,C 180,E1 -23016.036,E2 -23016.036} C_VEL
LIN {X 0,Y 393.103,Z 763.476,A -85,B 0,C 180,E1 -23016.692,E2 -23016.692} C_VEL
LIN {X 0,Y 395.96,Z 741.196,A -85,B 0,C 180,E1 -23017.111,E2 -23017.111} C_VEL
LIN {X 0,Y 411.562,Z 565.822,A -85,B 0,C 180,E1 -23019.885,E2 -23019.885} C_VEL
LIN {X 0,Y 410.414,Z 563.729,A -85,B 0,C 180,E1 -23020.439,E2 -23020.439} C_VEL
LIN {X 0,Y 408.494,Z 561.324,A -85,B 0,C 180,E1 -23021.349,E2 -23021.349} C_VEL
LIN {X 0,Y 404.965,Z 559.811,A -85,B 0,C 180,E1 -23022.997,E2 -23022.997} C_VEL
LIN {X 0,Y 401.883,Z 558.413,A -85,B 0,C 180,E1 -23024.608,E2 -23024.608} C_VEL
LIN {X 0,Y 400.917,Z 557.185,A -85,B 0,C 180,E1 -23025.209,E2 -23025.209} C_VEL
LIN {X 0,Y 397.429,Z 550.938,A -85,B 0,C 180,E1 -23027.799,E2 -23027.799} C_VEL
LIN {X 0,Y 394.489,Z 546.124,A -85,B 0,C 180,E1 -23030.517,E2 -23030.517} C_VEL
LIN {X 0,Y 392.148,Z 541.943,A -85,B 0,C 180,E1 -23033.558,E2 -23033.558} C_VEL
LIN {X 0,Y 390.288,Z 537.941,A -85,B 0,C 180,E1 -23039.853,E2 -23039.853} C_VEL
LIN {X 0,Y 392.508,Z 542.49,A -85,B 0,C 180,E1 -23046.656,E2 -23046.656} C_VEL
LIN {X 0,Y 395.375,Z 547.554,A -85,B 0,C 180,E1 -23050.05,E2 -23050.05} C_VEL
LIN {X 0,Y 397.98,Z 552.088,A -85,B 0,C 180,E1 -23052.331,E2 -23052.331} C_VEL
LIN {X 0,Y 401.863,Z 558.717,A -85,B 0,C 180,E1 -23055.071,E2 -23055.071} C_VEL
LIN {X 0,Y 404.374,Z 563.734,A -85,B 0,C 180,E1 -23056.631,E2 -23056.631} C_VEL
LIN {X 0,Y 408.397,Z 572.639,A -85,B 0,C 180,E1 -23058.885,E2 -23058.885} C_VEL
LIN {X 0,Y 391.606,Z 756.045,A -85,B 0,C 180,E1 -23061.775,E2 -23061.775} C_VEL
LIN {X 0,Y 387.504,Z 782.697,A -85,B 0,C 180,E1 -23062.31,E2 -23062.31} C_VEL
LIN {X 0,Y 382.937,Z 804.053,A -85,B 0,C 180,E1 -23062.857,E2 -23062.857} C_VEL
LIN {X 0,Y 376.571,Z 827.883,A -85,B 0,C 180,E1 -23063.643,E2 -23063.643} C_VEL
LIN {X 0,Y 369.944,Z 848.315,A -85,B 0,C 180,E1 -23064.5,E2 -23064.5} C_VEL
LIN {X 0,Y 361.635,Z 870.696,A -85,B 0,C 180,E1 -23065.662,E2 -23065.662} C_VEL
LIN {X 0,Y 352.221,Z 892.371,A -85,B 0,C 180,E1 -23067.083,E2 -23067.083} C_VEL
LIN {X 0,Y 342.489,Z 912.481,A -85,B 0,C 180,E1 -23068.681,E2 -23068.681} C_VEL
LIN {X 0,Y 331.792,Z 932.172,A -85,B 0,C 180,E1 -23070.617,E2 -23070.617} C_VEL
LIN {X 0,Y 321.761,Z 949.152,A -85,B 0,C 180,E1 -23072.632,E2 -23072.632} C_VEL
LIN {X 0,Y 309.321,Z 968.493,A -85,B 0,C 180,E1 -23075.452,E2 -23075.452} C_VEL
LIN {X 0,Y 298.879,Z 983.646,A -85,B 0,C 180,E1 -23078.169,E2 -23078.169} C_VEL
LIN {X 0,Y 286.971,Z 999.992,A -85,B 0,C 180,E1 -23081.786,E2 -23081.786} C_VEL
LIN {X 0,Y 277.221,Z 1012.838,A -85,B 0,C 180,E1 -23085.305,E2 -23085.305} C_VEL
LIN {X 0,Y 266.418,Z 1026.787,A -85,B 0,C 180,E1 -23090.075,E2 -23090.075} C_VEL
LIN {X 0,Y 258.816,Z 1036.675,A -85,B 0,C 180,E1 -23094.312,E2 -23094.312} C_VEL
LIN {X 0,Y 251.174,Z 1047.029,A -85,B 0,C 180,E1 -23099.895,E2 -23099.895} C_VEL
LIN {X 0,Y 246.334,Z 1054.194,A -85,B 0,C 180,E1 -23104.847,E2 -23104.847} C_VEL
LIN {X 0,Y 242.579,Z 1060.795,A -85,B 0,C 180,E1 -23110.746,E2 -23110.746} C_VEL
LIN {X 0,Y 240.805,Z 1064.907,A -85,B 0,C 180,E1 -23115.819,E2 -23115.819} C_VEL
LIN {X 0,Y 240.087,Z 1067.689,A -85,B 0,C 180,E1 -23120.652,E2 -23120.652} C_VEL
LIN {X 0,Y 239.978,Z 1069.439,A -85,B 0,C 180,E1 -23125.699,E2 -23125.699} C_VEL
LIN {X 0,Y 240.013,Z 1069.874,A -85,B 0,C 180,E1 -23130.477,E2 -23130.477} C_VEL
LIN {X 0,Y 239.979,Z 1069.146,A -85,B 0,C 180,E1 -23135.259,E2 -23135.259} C_VEL
LIN {X 0,Y 240.123,Z 1067.433,A -85,B 0,C 180,E1 -23139.83,E2 -23139.83} C_VEL
LIN {X 0,Y 240.923,Z 1064.548,A -85,B 0,C 180,E1 -23144.665,E2 -23144.665} C_VEL
LIN {X 0,Y 243.316,Z 1059.315,A -85,B 0,C 180,E1 -23150.696,E2 -23150.696} C_VEL
LIN {X 0,Y 246.977,Z 1053.117,A -85,B 0,C 180,E1 -23155.928,E2 -23155.928} C_VEL
LIN {X 0,Y 252.806,Z 1044.709,A -85,B 0,C 180,E1 -23161.472,E2 -23161.472} C_VEL
LIN {X 0,Y 259.86,Z 1035.189,A -85,B 0,C 180,E1 -23166.339,E2 -23166.339} C_VEL
LIN {X 0,Y 268.517,Z 1024.058,A -85,B 0,C 180,E1 -23170.948,E2 -23170.948} C_VEL
LIN {X 0,Y 278.183,Z 1011.425,A -85,B 0,C 180,E1 -23175.079,E2 -23175.079} C_VEL
LIN {X 0,Y 288.588,Z 997.719,A -85,B 0,C 180,E1 -23178.751,E2 -23178.751} C_VEL
LIN {X 0,Y 299.454,Z 982.611,A -85,B 0,C 180,E1 -23182,E2 -23182} C_VEL
LIN {X 0,Y 309.937,Z 967.357,A -85,B 0,C 180,E1 -23184.706,E2 -23184.706} C_VEL
LIN {X 0,Y 322.077,Z 948.345,A -85,B 0,C 180,E1 -23187.444,E2 -23187.444} C_VEL
LIN {X 0,Y 332.073,Z 931.362,A -85,B 0,C 180,E1 -23189.447,E2 -23189.447} C_VEL
LIN {X 0,Y 343.56,Z 909.916,A -85,B 0,C 180,E1 -23191.514,E2 -23191.514} C_VEL
LIN {X 0,Y 352.473,Z 891.385,A -85,B 0,C 180,E1 -23192.967,E2 -23192.967} C_VEL
LIN {X 0,Y 361.991,Z 869.216,A -85,B 0,C 180,E1 -23194.403,E2 -23194.403} C_VEL
LIN {X 0,Y 369.784,Z 848.163,A -85,B 0,C 180,E1 -23195.49,E2 -23195.49} C_VEL
LIN {X 0,Y 377.147,Z 825.318,A -85,B 0,C 180,E1 -23196.441,E2 -23196.441} C_VEL
LIN {X 0,Y 383.242,Z 801.786,A -85,B 0,C 180,E1 -23197.192,E2 -23197.192} C_VEL
LIN {X 0,Y 387.987,Z 779.065,A -85,B 0,C 180,E1 -23197.759,E2 -23197.759} C_VEL
LIN {X 0,Y 391.61,Z 753.921,A -85,B 0,C 180,E1 -23198.247,E2 -23198.247} C_VEL
LIN {X 0,Y 408.171,Z 572.362,A -85,B 0,C 180,E1 -23201.11,E2 -23201.11} C_VEL
LIN {X 0,Y 403.065,Z 561.18,A -85,B 0,C 180,E1 -23204.016,E2 -23204.016} C_VEL
LIN {X 0,Y 398.837,Z 553.773,A -85,B 0,C 180,E1 -23206.812,E2 -23206.812} C_VEL
LIN {X 0,Y 396.259,Z 549.369,A -85,B 0,C 180,E1 -23208.87,E2 -23208.87} C_VEL
LIN {X 0,Y 394.389,Z 546.098,A -85,B 0,C 180,E1 -23210.662,E2 -23210.662} C_VEL
LIN {X 0,Y 391.973,Z 541.841,A -85,B 0,C 180,E1 -23213.703,E2 -23213.703} C_VEL
LIN {X 0,Y 390.031,Z 537.096,A -85,B 0,C 180,E1 -23220.294,E2 -23220.294} C_VEL
LIN {X 0,Y 392.328,Z 542.451,A -85,B 0,C 180,E1 -23227.248,E2 -23227.248} C_VEL
LIN {X 0,Y 395.121,Z 547.368,A -85,B 0,C 180,E1 -23230.498,E2 -23230.498} C_VEL
LIN {X 0,Y 398.024,Z 552.338,A -85,B 0,C 180,E1 -23232.993,E2 -23232.993} C_VEL
LIN {X 0,Y 401.809,Z 558.914,A -85,B 0,C 180,E1 -23235.627,E2 -23235.627} C_VEL
LIN {X 0,Y 406.821,Z 568.129,A -85,B 0,C 180,E1 -23238.522,E2 -23238.522} C_VEL
LIN {X 0,Y 408.205,Z 570.909,A -85,B 0,C 180,E1 -23239.248,E2 -23239.248} C_VEL
LIN {X 0,Y 391.942,Z 748.124,A -85,B 0,C 180,E1 -23242.033,E2 -23242.033} C_VEL
LIN {X 0,Y 387.929,Z 774.587,A -85,B 0,C 180,E1 -23242.583,E2 -23242.583} C_VEL
LIN {X 0,Y 383.597,Z 795.382,A -85,B 0,C 180,E1 -23243.153,E2 -23243.153} C_VEL
LIN {X 0,Y 377.144,Z 820.112,A -85,B 0,C 180,E1 -23244.029,E2 -23244.029} C_VEL
LIN {X 0,Y 370.566,Z 840.752,A -85,B 0,C 180,E1 -23244.958,E2 -23244.958} C_VEL
LIN {X 0,Y 362.215,Z 863.439,A -85,B 0,C 180,E1 -23246.213,E2 -23246.213} C_VEL
LIN {X 0,Y 353.248,Z 884.154,A -85,B 0,C 180,E1 -23247.63,E2 -23247.63} C_VEL
LIN {X 0,Y 343.815,Z 903.806,A -85,B 0,C 180,E1 -23249.254,E2 -23249.254} C_VEL
LIN {X 0,Y 333.244,Z 923.3,A -85,B 0,C 180,E1 -23251.226,E2 -23251.226} C_VEL
LIN {X 0,Y 323.411,Z 939.944,A -85,B 0,C 180,E1 -23253.248,E2 -23253.248} C_VEL
LIN {X 0,Y 311.444,Z 958.487,A -85,B 0,C 180,E1 -23255.997,E2 -23255.997} C_VEL
LIN {X 0,Y 301.096,Z 973.388,A -85,B 0,C 180,E1 -23258.703,E2 -23258.703} C_VEL
LIN {X 0,Y 289.24,Z 989.443,A -85,B 0,C 180,E1 -23262.287,E2 -23262.287} C_VEL
LIN {X 0,Y 279.959,Z 1001.417,A -85,B 0,C 180,E1 -23265.587,E2 -23265.587} C_VEL
LIN {X 0,Y 269.899,Z 1014.105,A -85,B 0,C 180,E1 -23269.863,E2 -23269.863} C_VEL
LIN {X 0,Y 261.604,Z 1024.322,A -85,B 0,C 180,E1 -23274.212,E2 -23274.212} C_VEL
LIN {X 0,Y 254.126,Z 1033.856,A -85,B 0,C 180,E1 -23279.236,E2 -23279.236} C_VEL
LIN {X 0,Y 248.351,Z 1041.457,A -85,B 0,C 180,E1 -23284.482,E2 -23284.482} C_VEL
LIN {X 0,Y 244.263,Z 1047.581,A -85,B 0,C 180,E1 -23289.888,E2 -23289.888} C_VEL
LIN {X 0,Y 241.629,Z 1052.21,A -85,B 0,C 180,E1 -23295.624,E2 -23295.624} C_VEL
LIN {X 0,Y 240.529,Z 1054.881,A -85,B 0,C 180,E1 -23300.429,E2 -23300.429} C_VEL
LIN {X 0,Y 240.092,Z 1056.571,A -85,B 0,C 180,E1 -23305.462,E2 -23305.462} C_VEL
LIN {X 0,Y 240.019,Z 1057.048,A -85,B 0,C 180,E1 -23310.716,E2 -23310.716} C_VEL
LIN {X 0,Y 240.128,Z 1056.345,A -85,B 0,C 180,E1 -23315.496,E2 -23315.496} C_VEL
LIN {X 0,Y 240.584,Z 1054.724,A -85,B 0,C 180,E1 -23320.053,E2 -23320.053} C_VEL
LIN {X 0,Y 241.853,Z 1051.833,A -85,B 0,C 180,E1 -23325.098,E2 -23325.098} C_VEL
LIN {X 0,Y 244.807,Z 1046.725,A -85,B 0,C 180,E1 -23331.065,E2 -23331.065} C_VEL
LIN {X 0,Y 248.719,Z 1041.028,A -85,B 0,C 180,E1 -23335.989,E2 -23335.989} C_VEL
LIN {X 0,Y 254.913,Z 1032.891,A -85,B 0,C 180,E1 -23341.446,E2 -23341.446} C_VEL
LIN {X 0,Y 261.857,Z 1024.11,A -85,B 0,C 180,E1 -23346.018,E2 -23346.018} C_VEL
LIN {X 0,Y 270.636,Z 1013.349,A -85,B 0,C 180,E1 -23350.56,E2 -23350.56} C_VEL
LIN {X 0,Y 280.339,Z 1001.082,A -85,B 0,C 180,E1 -23354.64,E2 -23354.64} C_VEL
LIN {X 0,Y 290.727,Z 987.727,A -85,B 0,C 180,E1 -23358.273,E2 -23358.273} C_VEL
LIN {X 0,Y 301.534,Z 972.984,A -85,B 0,C 180,E1 -23361.498,E2 -23361.498} C_VEL
LIN {X 0,Y 311.285,Z 958.956,A -85,B 0,C 180,E1 -23364.043,E2 -23364.043} C_VEL
LIN {X 0,Y 323.34,Z 940.357,A -85,B 0,C 180,E1 -23366.814,E2 -23366.814} C_VEL
LIN {X 0,Y 333.084,Z 923.911,A -85,B 0,C 180,E1 -23368.82,E2 -23368.82} C_VEL
LIN {X 0,Y 343.656,Z 904.542,A -85,B 0,C 180,E1 -23370.794,E2 -23370.794} C_VEL
LIN {X 0,Y 353.085,Z 884.958,A -85,B 0,C 180,E1 -23372.421,E2 -23372.421} C_VEL
LIN {X 0,Y 361.674,Z 865.211,A -85,B 0,C 180,E1 -23373.782,E2 -23373.782} C_VEL
LIN {X 0,Y 370.027,Z 842.972,A -85,B 0,C 180,E1 -23375.038,E2 -23375.038} C_VEL
LIN {X 0,Y 376.604,Z 822.634,A -85,B 0,C 180,E1 -23375.969,E2 -23375.969} C_VEL
LIN {X 0,Y 383.142,Z 798.421,A -85,B 0,C 180,E1 -23376.856,E2 -23376.856} C_VEL
LIN {X 0,Y 387.721,Z 776.866,A -85,B 0,C 180,E1 -23377.465,E2 -23377.465} C_VEL
LIN {X 0,Y 391.694,Z 752.46,A -85,B 0,C 180,E1 -23377.997,E2 -23377.997} C_VEL
LIN {X 0,Y 396.631,Z 700.921,A -85,B 0,C 180,E1 -23378.831,E2 -23378.831} C_VEL
LIN {X 0,Y 408.39,Z 570.784,A -85,B 0,C 180,E1 -23380.885,E2 -23380.885} C_VEL
LIN {X 0,Y 403.478,Z 561.727,A -85,B 0,C 180,E1 -23383.59,E2 -23383.59} C_VEL
LIN {X 0,Y 400.917,Z 557.185,A -85,B 0,C 180,E1 -23385.209,E2 -23385.209} C_VEL
LIN {X 0,Y 399.374,Z 555.683,A -85,B 0,C 180,E1 -23386.195,E2 -23386.195} C_VEL
LIN {X 0,Y 396.403,Z 555.775,A -85,B 0,C 180,E1 -23388.086,E2 -23388.086} C_VEL
LIN {X 0,Y 394.402,Z 555.502,A -85,B 0,C 180,E1 -23389.605,E2 -23389.605} C_VEL
LIN {X 0,Y 393.763,Z 554.568,A -85,B 0,C 180,E1 -23390.233,E2 -23390.233} C_VEL
LIN {X 0,Y 391.077,Z 549.826,A -85,B 0,C 180,E1 -23393.688,E2 -23393.688} C_VEL
LIN {X 0,Y 389.312,Z 545.893,A -85,B 0,C 180,E1 -23399.853,E2 -23399.853} C_VEL
LIN {X 0,Y 391.38,Z 550.298,A -85,B 0,C 180,E1 -23406.454,E2 -23406.454} C_VEL
LIN {X 0,Y 394.095,Z 555.245,A -85,B 0,C 180,E1 -23409.787,E2 -23409.787} C_VEL
LIN {X 0,Y 396.713,Z 559.961,A -85,B 0,C 180,E1 -23412.149,E2 -23412.149} C_VEL
LIN {X 0,Y 400.42,Z 566.488,A -85,B 0,C 180,E1 -23414.83,E2 -23414.83} C_VEL
LIN {X 0,Y 402.815,Z 571.498,A -85,B 0,C 180,E1 -23416.364,E2 -23416.364} C_VEL
LIN {X 0,Y 405.394,Z 577.486,A -85,B 0,C 180,E1 -23417.889,E2 -23417.889} C_VEL
LIN {X 0,Y 388.699,Z 755.851,A -85,B 0,C 180,E1 -23420.676,E2 -23420.676} C_VEL
LIN {X 0,Y 384.54,Z 782.432,A -85,B 0,C 180,E1 -23421.202,E2 -23421.202} C_VEL
LIN {X 0,Y 379.886,Z 803.848,A -85,B 0,C 180,E1 -23421.739,E2 -23421.739} C_VEL
LIN {X 0,Y 373.004,Z 828.963,A -85,B 0,C 180,E1 -23422.559,E2 -23422.559} C_VEL
LIN {X 0,Y 366.53,Z 848.493,A -85,B 0,C 180,E1 -23423.369,E2 -23423.369} C_VEL
LIN {X 0,Y 358.2,Z 870.486,A -85,B 0,C 180,E1 -23424.494,E2 -23424.494} C_VEL
LIN {X 0,Y 348.495,Z 892.373,A -85,B 0,C 180,E1 -23425.909,E2 -23425.909} C_VEL
LIN {X 0,Y 338.281,Z 913.007,A -85,B 0,C 180,E1 -23427.534,E2 -23427.534} C_VEL
LIN {X 0,Y 327.279,Z 932.677,A -85,B 0,C 180,E1 -23429.464,E2 -23429.464} C_VEL
LIN {X 0,Y 316.723,Z 950.054,A -85,B 0,C 180,E1 -23431.527,E2 -23431.527} C_VEL
LIN {X 0,Y 304.621,Z 968.276,A -85,B 0,C 180,E1 -23434.191,E2 -23434.191} C_VEL
LIN {X 0,Y 294.465,Z 982.575,A -85,B 0,C 180,E1 -23436.739,E2 -23436.739} C_VEL
LIN {X 0,Y 282.648,Z 998.356,A -85,B 0,C 180,E1 -23440.171,E2 -23440.171} C_VEL
LIN {X 0,Y 272.404,Z 1011.332,A -85,B 0,C 180,E1 -23443.688,E2 -23443.688} C_VEL
LIN {X 0,Y 262.32,Z 1023.944,A -85,B 0,C 180,E1 -23447.866,E2 -23447.866} C_VEL
LIN {X 0,Y 253.234,Z 1035.055,A -85,B 0,C 180,E1 -23452.55,E2 -23452.55} C_VEL
LIN {X 0,Y 245.787,Z 1044.568,A -85,B 0,C 180,E1 -23457.521,E2 -23457.521} C_VEL
LIN {X 0,Y 239.583,Z 1052.955,A -85,B 0,C 180,E1 -23463.209,E2 -23463.209} C_VEL
LIN {X 0,Y 235.65,Z 1059.142,A -85,B 0,C 180,E1 -23468.598,E2 -23468.598} C_VEL
LIN {X 0,Y 233.042,Z 1064.36,A -85,B 0,C 180,E1 -23474.827,E2 -23474.827} C_VEL
LIN {X 0,Y 232.155,Z 1067.239,A -85,B 0,C 180,E1 -23479.829,E2 -23479.829} C_VEL
LIN {X 0,Y 231.979,Z 1068.975,A -85,B 0,C 180,E1 -23484.669,E2 -23484.669} C_VEL
LIN {X 0,Y 232.016,Z 1069.664,A -85,B 0,C 180,E1 -23489.506,E2 -23489.506} C_VEL
LIN {X 0,Y 231.98,Z 1069.213,A -85,B 0,C 180,E1 -23494.45,E2 -23494.45} C_VEL
LIN {X 0,Y 232.109,Z 1067.452,A -85,B 0,C 180,E1 -23499.672,E2 -23499.672} C_VEL
LIN {X 0,Y 232.91,Z 1064.66,A -85,B 0,C 180,E1 -23504.672,E2 -23504.672} C_VEL
LIN {X 0,Y 235.1,Z 1060.113,A -85,B 0,C 180,E1 -23510.411,E2 -23510.411} C_VEL
LIN {X 0,Y 239.15,Z 1053.516,A -85,B 0,C 180,E1 -23516.307,E2 -23516.307} C_VEL
LIN {X 0,Y 244.601,Z 1046.017,A -85,B 0,C 180,E1 -23521.55,E2 -23521.55} C_VEL
LIN {X 0,Y 252.112,Z 1036.366,A -85,B 0,C 180,E1 -23526.789,E2 -23526.789} C_VEL
LIN {X 0,Y 260.13,Z 1026.429,A -85,B 0,C 180,E1 -23531.115,E2 -23531.115} C_VEL
LIN {X 0,Y 271.006,Z 1012.96,A -85,B 0,C 180,E1 -23535.787,E2 -23535.787} C_VEL
LIN {X 0,Y 280.947,Z 1000.332,A -85,B 0,C 180,E1 -23539.294,E2 -23539.294} C_VEL
LIN {X 0,Y 293.219,Z 984.095,A -85,B 0,C 180,E1 -23542.934,E2 -23542.934} C_VEL
LIN {X 0,Y 303.947,Z 969.002,A -85,B 0,C 180,E1 -23545.66,E2 -23545.66} C_VEL
LIN {X 0,Y 316.013,Z 950.918,A -85,B 0,C 180,E1 -23548.335,E2 -23548.335} C_VEL
LIN {X 0,Y 326.55,Z 933.59,A -85,B 0,C 180,E1 -23550.412,E2 -23550.412} C_VEL
LIN {X 0,Y 337.512,Z 914.075,A -85,B 0,C 180,E1 -23552.35,E2 -23552.35} C_VEL
